LIN {X 0,Y 464.537,Z 936.315,A -85,B 0,C 180,E1 20832.687,E2 20832.687} C_VEL
LIN {X 0,Y 462.076,Z 957.618,A -85,B 0,C 180,E1 20831.71,E2 20831.71} C_VEL
LIN {X 0,Y 459.345,Z 978.775,A -85,B 0,C 180,E1 20830.531,E2 20830.531} C_VEL
LIN {X 0,Y 456.263,Z 999.373,A -85,B 0,C 180,E1 20829.127,E2 20829.127} C_VEL
LIN {X 0,Y 453.115,Z 1019.391,A -85,B 0,C 180,E1 20827.519,E2 20827.519} C_VEL
LIN {X 0,Y 449.993,Z 1037.958,A -85,B 0,C 180,E1 20825.758,E2 20825.758} C_VEL
LIN {X 0,Y 446.561,Z 1057.743,A -85,B 0,C 180,E1 20823.576,E2 20823.576} C_VEL
LIN {X 0,Y 443.731,Z 1074.21,A -85,B 0,C 180,E1 20821.464,E2 20821.464} C_VEL
LIN {X 0,Y 440.916,Z 1090.601,A -85,B 0,C 180,E1 20819.031,E2 20819.031} C_VEL
LIN {X 0,Y 438.586,Z 1105.226,A -85,B 0,C 180,E1 20816.54,E2 20816.54} C_VEL
LIN {X 0,Y 436.583,Z 1118.418,A -85,B 0,C 180,E1 20813.914,E2 20813.914} C_VEL
LIN {X 0,Y 434.957,Z 1130.257,A -85,B 0,C 180,E1 20811.156,E2 20811.156} C_VEL
LIN {X 0,Y 433.707,Z 1140.6,A -85,B 0,C 180,E1 20808.272,E2 20808.272} C_VEL
LIN {X 0,Y 432.808,Z 1149.992,A -85,B 0,C 180,E1 20805.132,E2 20805.132} C_VEL
LIN {X 0,Y 432.328,Z 1156.56,A -85,B 0,C 180,E1 20802.42,E2 20802.42} C_VEL
LIN {X 0,Y 432.052,Z 1162.429,A -85,B 0,C 180,E1 20799.322,E2 20799.322} C_VEL
LIN {X 0,Y 431.943,Z 1166.119,A -85,B 0,C 180,E1 20796.646,E2 20796.646} C_VEL
LIN {X 0,Y 431.895,Z 1168.848,A -85,B 0,C 180,E1 20793.583,E2 20793.583} C_VEL
LIN {X 0,Y 431.889,Z 1169.849,A -85,B 0,C 180,E1 20790.928,E2 20790.928} C_VEL
LIN {X 0,Y 431.905,Z 1169.689,A -85,B 0,C 180,E1 20788.142,E2 20788.142} C_VEL
LIN {X 0,Y 431.913,Z 1167.954,A -85,B 0,C 180,E1 20785.219,E2 20785.219} C_VEL
LIN {X 0,Y 431.957,Z 1165,A -85,B 0,C 180,E1 20782.418,E2 20782.418} C_VEL
LIN {X 0,Y 432.148,Z 1160.081,A -85,B 0,C 180,E1 20779.333,E2 20779.333} C_VEL
LIN {X 0,Y 432.493,Z 1154.133,A -85,B 0,C 180,E1 20776.497,E2 20776.497} C_VEL
LIN {X 0,Y 433.141,Z 1146.144,A -85,B 0,C 180,E1 20773.505,E2 20773.505} C_VEL
LIN {X 0,Y 434.129,Z 1136.928,A -85,B 0,C 180,E1 20770.631,E2 20770.631} C_VEL
LIN {X 0,Y 435.547,Z 1125.712,A -85,B 0,C 180,E1 20767.741,E2 20767.741} C_VEL
LIN {X 0,Y 437.273,Z 1113.83,A -85,B 0,C 180,E1 20765.119,E2 20765.119} C_VEL
LIN {X 0,Y 439.435,Z 1099.732,A -85,B 0,C 180,E1 20762.49,E2 20762.49} C_VEL
LIN {X 0,Y 442.212,Z 1082.982,A -85,B 0,C 180,E1 20759.795,E2 20759.795} C_VEL
LIN {X 0,Y 445.049,Z 1066.635,A -85,B 0,C 180,E1 20757.524,E2 20757.524} C_VEL
LIN {X 0,Y 448.073,Z 1049.082,A -85,B 0,C 180,E1 20755.427,E2 20755.427} C_VEL
LIN {X 0,Y 451.263,Z 1030.575,A -85,B 0,C 180,E1 20753.501,E2 20753.501} C_VEL
LIN {X 0,Y 454.405,Z 1011.335,A -85,B 0,C 180,E1 20751.807,E2 20751.807} C_VEL
LIN {X 0,Y 457.549,Z 991.207,A -85,B 0,C 180,E1 20750.282,E2 20750.282} C_VEL
LIN {X 0,Y 460.346,Z 970.958,A -85,B 0,C 180,E1 20749.009,E2 20749.009} C_VEL
LIN {X 0,Y 463.115,Z 948.971,A -85,B 0,C 180,E1 20747.862,E2 20747.862} C_VEL
LIN {X 0,Y 465.361,Z 927.596,A -85,B 0,C 180,E1 20746.986,E2 20746.986} C_VEL
LIN {X 0,Y 467.381,Z 903.992,A -85,B 0,C 180,E1 20746.249,E2 20746.249} C_VEL
LIN {X 0,Y 468.614,Z 882.183,A -85,B 0,C 180,E1 20745.765,E2 20745.765} C_VEL
LIN {X 0,Y 474.642,Z 683.276,A -85,B 0,C 180,E1 20742.249,E2 20742.249} C_VEL
LIN {X 0,Y 477.34,Z 594.822,A -85,B 0,C 180,E1 20740.649,E2 20740.649} C_VEL
LIN {X 0,Y 465.354,Z 575.94,A -85,B 0,C 180,E1 20738.463,E2 20738.463} C_VEL
LIN {X 0,Y 455.422,Z 561.586,A -85,B 0,C 180,E1 20736.51,E2 20736.51} C_VEL
LIN {X 0,Y 446.552,Z 549.244,A -85,B 0,C 180,E1 20734.622,E2 20734.622} C_VEL
LIN {X 0,Y 442.442,Z 543.776,A -85,B 0,C 180,E1 20733.696,E2 20733.696} C_VEL
LIN {X 0,Y 438.178,Z 538.303,A -85,B 0,C 180,E1 20732.699,E2 20732.699} C_VEL
LIN {X 0,Y 436.612,Z 536.106,A -85,B 0,C 180,E1 20732.247,E2 20732.247} C_VEL
LIN {X 0,Y 435.538,Z 533.777,A -85,B 0,C 180,E1 20731.716,E2 20731.716} C_VEL
LIN {X 0,Y 433.709,Z 530.877,A -85,B 0,C 180,E1 20730.937,E2 20730.937} C_VEL
LIN {X 0,Y 433.24,Z 529.049,A -85,B 0,C 180,E1 20730.552,E2 20730.552} C_VEL
LIN {X 0,Y 433.259,Z 529.072,A -85,B 0,C 180,E1 20726.892,E2 20726.892} C_VEL
LIN {X 0,Y 433.245,Z 529.031,A -85,B 0,C 180,E1 20723.099,E2 20723.099} C_VEL
LIN {X 0,Y 433.233,Z 529.057,A -85,B 0,C 180,E1 20719.41,E2 20719.41} C_VEL
LIN {X 0,Y 433.242,Z 529.06,A -85,B 0,C 180,E1 20715.528,E2 20715.528} C_VEL
LIN {X 0,Y 433.249,Z 529.036,A -85,B 0,C 180,E1 20711.852,E2 20711.852} C_VEL
LIN {X 0,Y 433.249,Z 529.074,A -85,B 0,C 180,E1 20708.083,E2 20708.083} C_VEL
LIN {X 0,Y 433.252,Z 529.078,A -85,B 0,C 180,E1 20704.235,E2 20704.235} C_VEL
LIN {X 0,Y 433.254,Z 529.079,A -85,B 0,C 180,E1 20700.396,E2 20700.396} C_VEL
LIN {X 0,Y 433.255,Z 529.08,A -85,B 0,C 180,E1 20696.56,E2 20696.56} C_VEL
LIN {X 0,Y 433.254,Z 529.079,A -85,B 0,C 180,E1 20692.708,E2 20692.708} C_VEL
LIN {X 0,Y 433.225,Z 529.03,A -85,B 0,C 180,E1 20688.956,E2 20688.956} C_VEL
LIN {X 0,Y 433.233,Z 529.076,A -85,B 0,C 180,E1 20685.156,E2 20685.156} C_VEL
LIN {X 0,Y 433.249,Z 529.036,A -85,B 0,C 180,E1 20681.429,E2 20681.429} C_VEL
LIN {X 0,Y 433.262,Z 529.045,A -85,B 0,C 180,E1 20677.618,E2 20677.618} C_VEL
LIN {X 0,Y 433.23,Z 529.076,A -85,B 0,C 180,E1 20673.844,E2 20673.844} C_VEL
LIN {X 0,Y 433.205,Z 529.041,A -85,B 0,C 180,E1 20670.096,E2 20670.096} C_VEL
LIN {X 0,Y 433.235,Z 529.287,A -85,B 0,C 180,E1 20668.028,E2 20668.028} C_VEL
LIN {X 0,Y 434.286,Z 532.203,A -85,B 0,C 180,E1 20667.715,E2 20667.715} C_VEL
LIN {X 0,Y 436.698,Z 534.701,A -85,B 0,C 180,E1 20667.137,E2 20667.137} C_VEL
LIN {X 0,Y 438.011,Z 535.73,A -85,B 0,C 180,E1 20666.838,E2 20666.838} C_VEL
LIN {X 0,Y 440.301,Z 539.399,A -85,B 0,C 180,E1 20666.274,E2 20666.274} C_VEL
LIN {X 0,Y 442.889,Z 541.924,A -85,B 0,C 180,E1 20665.698,E2 20665.698} C_VEL
LIN {X 0,Y 446.059,Z 546.162,A -85,B 0,C 180,E1 20664.982,E2 20664.982} C_VEL
LIN {X 0,Y 447.716,Z 548.187,A -85,B 0,C 180,E1 20664.622,E2 20664.622} C_VEL
LIN {X 0,Y 452.356,Z 554.185,A -85,B 0,C 180,E1 20663.635,E2 20663.635} C_VEL
LIN {X 0,Y 459.599,Z 563.567,A -85,B 0,C 180,E1 20662.177,E2 20662.177} C_VEL
LIN {X 0,Y 471.372,Z 579.87,A -85,B 0,C 180,E1 20659.97,E2 20659.97} C_VEL
LIN {X 0,Y 477.284,Z 588.789,A -85,B 0,C 180,E1 20658.922,E2 20658.922} C_VEL
LIN {X 0,Y 470.626,Z 800.468,A -85,B 0,C 180,E1 20655.158,E2 20655.158} C_VEL
LIN {X 0,Y 469.076,Z 852.641,A -85,B 0,C 180,E1 20654.242,E2 20654.242} C_VEL
LIN {X 0,Y 468.06,Z 860.337,A -85,B 0,C 180,E1 20654.186,E2 20654.186} C_VEL
LIN {X 0,Y 462.56,Z 879.729,A -85,B 0,C 180,E1 20654.257,E2 20654.257} C_VEL
LIN {X 0,Y 461.266,Z 887.24,A -85,B 0,C 180,E1 20654.119,E2 20654.119} C_VEL
LIN {X 0,Y 459.307,Z 908.693,A -85,B 0,C 180,E1 20653.361,E2 20653.361} C_VEL
LIN {X 0,Y 456.826,Z 930.04,A -85,B 0,C 180,E1 20652.387,E2 20652.387} C_VEL
LIN {X 0,Y 454.256,Z 949.055,A -85,B 0,C 180,E1 20651.325,E2 20651.325} C_VEL
LIN {X 0,Y 450.888,Z 970.761,A -85,B 0,C 180,E1 20649.857,E2 20649.857} C_VEL
LIN {X 0,Y 447.634,Z 990.006,A -85,B 0,C 180,E1 20648.305,E2 20648.305} C_VEL
LIN {X 0,Y 444.229,Z 1008.539,A -85,B 0,C 180,E1 20646.532,E2 20646.532} C_VEL
LIN {X 0,Y 440.839,Z 1026.51,A -85,B 0,C 180,E1 20644.543,E2 20644.543} C_VEL
LIN {X 0,Y 437.473,Z 1043.473,A -85,B 0,C 180,E1 20642.332,E2 20642.332} C_VEL
LIN {X 0,Y 434.444,Z 1059.247,A -85,B 0,C 180,E1 20639.962,E2 20639.962} C_VEL
LIN {X 0,Y 431.785,Z 1073.227,A -85,B 0,C 180,E1 20637.515,E2 20637.515} C_VEL
LIN {X 0,Y 429.287,Z 1087.359,A -85,B 0,C 180,E1 20634.64,E2 20634.64} C_VEL
LIN {X 0,Y 427.514,Z 1098.552,A -85,B 0,C 180,E1 20631.976,E2 20631.976} C_VEL
LIN {X 0,Y 425.953,Z 1109.995,A -85,B 0,C 180,E1 20628.759,E2 20628.759} C_VEL
LIN {X 0,Y 425.007,Z 1118.9,A -85,B 0,C 180,E1 20625.803,E2 20625.803} C_VEL
LIN {X 0,Y 424.409,Z 1125.853,A -85,B 0,C 180,E1 20622.933,E2 20622.933} C_VEL
LIN {X 0,Y 424.087,Z 1131.521,A -85,B 0,C 180,E1 20620.048,E2 20620.048} C_VEL
LIN {X 0,Y 423.938,Z 1135.585,A -85,B 0,C 180,E1 20617.181,E2 20617.181} C_VEL
LIN {X 0,Y 423.914,Z 1138.257,A -85,B 0,C 180,E1 20614.464,E2 20614.464} C_VEL
LIN {X 0,Y 423.907,Z 1139.772,A -85,B 0,C 180,E1 20611.352,E2 20611.352} C_VEL
LIN {X 0,Y 423.905,Z 1139.788,A -85,B 0,C 180,E1 20608.649,E2 20608.649} C_VEL
LIN {X 0,Y 423.911,Z 1138.333,A -85,B 0,C 180,E1 20605.536,E2 20605.536} C_VEL
LIN {X 0,Y 423.935,Z 1135.693,A -85,B 0,C 180,E1 20602.819,E2 20602.819} C_VEL
LIN {X 0,Y 424.081,Z 1131.671,A -85,B 0,C 180,E1 20599.952,E2 20599.952} C_VEL
LIN {X 0,Y 424.401,Z 1126.052,A -85,B 0,C 180,E1 20597.067,E2 20597.067} C_VEL
LIN {X 0,Y 425.034,Z 1118.689,A -85,B 0,C 180,E1 20594.024,E2 20594.024} C_VEL
LIN {X 0,Y 425.988,Z 1109.72,A -85,B 0,C 180,E1 20591.068,E2 20591.068} C_VEL
LIN {X 0,Y 427.62,Z 1097.777,A -85,B 0,C 180,E1 20587.742,E2 20587.742} C_VEL
LIN {X 0,Y 429.442,Z 1086.497,A -85,B 0,C 180,E1 20585.076,E2 20585.076} C_VEL
LIN {X 0,Y 431.907,Z 1072.551,A -85,B 0,C 180,E1 20582.27,E2 20582.27} C_VEL
LIN {X 0,Y 434.689,Z 1058.071,A -85,B 0,C 180,E1 20579.753,E2 20579.753} C_VEL
LIN {X 0,Y 437.749,Z 1042.06,A -85,B 0,C 180,E1 20577.381,E2 20577.381} C_VEL
LIN {X 0,Y 441.243,Z 1024.324,A -85,B 0,C 180,E1 20575.114,E2 20575.114} C_VEL
LIN {X 0,Y 444.47,Z 1007.272,A -85,B 0,C 180,E1 20573.246,E2 20573.246} C_VEL
LIN {X 0,Y 448.168,Z 986.861,A -85,B 0,C 180,E1 20571.338,E2 20571.338} C_VEL
LIN {X 0,Y 451.394,Z 967.84,A -85,B 0,C 180,E1 20569.835,E2 20569.835} C_VEL
LIN {X 0,Y 454.551,Z 946.907,A -85,B 0,C 180,E1 20568.456,E2 20568.456} C_VEL
LIN {X 0,Y 457.149,Z 927.589,A -85,B 0,C 180,E1 20567.396,E2 20567.396} C_VEL
LIN {X 0,Y 459.664,Z 904.799,A -85,B 0,C 180,E1 20566.396,E2 20566.396} C_VEL
LIN {X 0,Y 461.729,Z 881.961,A -85,B 0,C 180,E1 20565.628,E2 20565.628} C_VEL
LIN {X 0,Y 463.1,Z 859.095,A -85,B 0,C 180,E1 20565.097,E2 20565.097} C_VEL
LIN {X 0,Y 469.617,Z 660.74,A -85,B 0,C 180,E1 20561.547,E2 20561.547} C_VEL
LIN {X 0,Y 471.884,Z 592.324,A -85,B 0,C 180,E1 20560.3,E2 20560.3} C_VEL
LIN {X 0,Y 459.321,Z 574.267,A -85,B 0,C 180,E1 20557.949,E2 20557.949} C_VEL
LIN {X 0,Y 450.693,Z 562.894,A -85,B 0,C 180,E1 20556.205,E2 20556.205} C_VEL
LIN {X 0,Y 446.573,Z 557.588,A -85,B 0,C 180,E1 20555.325,E2 20555.325} C_VEL
LIN {X 0,Y 442.923,Z 552.874,A -85,B 0,C 180,E1 20554.514,E2 20554.514} C_VEL
LIN {X 0,Y 438.984,Z 547.828,A -85,B 0,C 180,E1 20553.606,E2 20553.606} C_VEL
LIN {X 0,Y 435.708,Z 543.956,A -85,B 0,C 180,E1 20552.83,E2 20552.83} C_VEL
LIN {X 0,Y 434.421,Z 542.142,A -85,B 0,C 180,E1 20552.508,E2 20552.508} C_VEL
LIN {X 0,Y 431.434,Z 539.099,A -85,B 0,C 180,E1 20551.78,E2 20551.78} C_VEL
LIN {X 0,Y 429.779,Z 536.292,A -85,B 0,C 180,E1 20551.33,E2 20551.33} C_VEL
LIN {X 0,Y 426.843,Z 533.857,A -85,B 0,C 180,E1 20550.591,E2 20550.591} C_VEL
LIN {X 0,Y 425.447,Z 530.984,A -85,B 0,C 180,E1 20550.173,E2 20550.173} C_VEL
LIN {X 0,Y 425.266,Z 530.032,A -85,B 0,C 180,E1 20550.092,E2 20550.092} C_VEL
LIN {X 0,Y 425.304,Z 530.071,A -85,B 0,C 180,E1 20546.38,E2 20546.38} C_VEL
LIN {X 0,Y 425.32,Z 530.023,A -85,B 0,C 180,E1 20542.5,E2 20542.5} C_VEL
LIN {X 0,Y 425.295,Z 530.039,A -85,B 0,C 180,E1 20538.789,E2 20538.789} C_VEL
LIN {X 0,Y 425.283,Z 530.05,A -85,B 0,C 180,E1 20534.988,E2 20534.988} C_VEL
LIN {X 0,Y 425.29,Z 530.064,A -85,B 0,C 180,E1 20531.115,E2 20531.115} C_VEL
LIN {X 0,Y 425.312,Z 530.065,A -85,B 0,C 180,E1 20527.294,E2 20527.294} C_VEL
LIN {X 0,Y 425.316,Z 530.066,A -85,B 0,C 180,E1 20523.505,E2 20523.505} C_VEL
LIN {X 0,Y 425.318,Z 530.068,A -85,B 0,C 180,E1 20519.596,E2 20519.596} C_VEL
LIN {X 0,Y 425.314,Z 530.071,A -85,B 0,C 180,E1 20515.686,E2 20515.686} C_VEL
LIN {X 0,Y 425.313,Z 530.068,A -85,B 0,C 180,E1 20511.778,E2 20511.778} C_VEL
LIN {X 0,Y 425.306,Z 530.02,A -85,B 0,C 180,E1 20507.923,E2 20507.923} C_VEL
LIN {X 0,Y 425.314,Z 530.047,A -85,B 0,C 180,E1 20504.175,E2 20504.175} C_VEL
LIN {X 0,Y 425.3,Z 530.048,A -85,B 0,C 180,E1 20500.356,E2 20500.356} C_VEL
LIN {X 0,Y 425.291,Z 530.026,A -85,B 0,C 180,E1 20496.475,E2 20496.475} C_VEL
LIN {X 0,Y 425.308,Z 530.055,A -85,B 0,C 180,E1 20492.703,E2 20492.703} C_VEL
LIN {X 0,Y 425.34,Z 530.158,A -85,B 0,C 180,E1 20491.037,E2 20491.037} C_VEL
LIN {X 0,Y 426.673,Z 533.637,A -85,B 0,C 180,E1 20490.212,E2 20490.212} C_VEL
LIN {X 0,Y 428.26,Z 535.701,A -85,B 0,C 180,E1 20489.561,E2 20489.561} C_VEL
LIN {X 0,Y 431.136,Z 539.923,A -85,B 0,C 180,E1 20488.742,E2 20488.742} C_VEL
LIN {X 0,Y 433.347,Z 542.697,A -85,B 0,C 180,E1 20488.183,E2 20488.183} C_VEL
LIN {X 0,Y 437.254,Z 547.799,A -85,B 0,C 180,E1 20487.224,E2 20487.224} C_VEL
LIN {X 0,Y 441.264,Z 553.084,A -85,B 0,C 180,E1 20486.28,E2 20486.28} C_VEL
LIN {X 0,Y 450.845,Z 566.205,A -85,B 0,C 180,E1 20484.163,E2 20484.163} C_VEL
LIN {X 0,Y 462.48,Z 583.389,A -85,B 0,C 180,E1 20481.807,E2 20481.807} C_VEL
LIN {X 0,Y 472.123,Z 598.819,A -85,B 0,C 180,E1 20479.998,E2 20479.998} C_VEL
LIN {X 0,Y 465.354,Z 804.742,A -85,B 0,C 180,E1 20476.303,E2 20476.303} C_VEL
LIN {X 0,Y 462.484,Z 890.625,A -85,B 0,C 180,E1 20474.758,E2 20474.758} C_VEL
LIN {X 0,Y 460.703,Z 913.95,A -85,B 0,C 180,E1 20474.154,E2 20474.154} C_VEL
LIN {X 0,Y 458.512,Z 936.783,A -85,B 0,C 180,E1 20473.343,E2 20473.343} C_VEL
LIN {X 0,Y 456,Z 957.431,A -85,B 0,C 180,E1 20472.387,E2 20472.387} C_VEL
LIN {X 0,Y 453.13,Z 978.557,A -85,B 0,C 180,E1 20471.199,E2 20471.199} C_VEL
LIN {X 0,Y 449.911,Z 998.994,A -85,B 0,C 180,E1 20469.794,E2 20469.794} C_VEL
LIN {X 0,Y 446.561,Z 1019.08,A -85,B 0,C 180,E1 20468.168,E2 20468.168} C_VEL
LIN {X 0,Y 443.253,Z 1037.646,A -85,B 0,C 180,E1 20466.388,E2 20466.388} C_VEL
LIN {X 0,Y 439.617,Z 1057.429,A -85,B 0,C 180,E1 20464.178,E2 20464.178} C_VEL
LIN {X 0,Y 436.566,Z 1074.041,A -85,B 0,C 180,E1 20462.019,E2 20462.019} C_VEL
LIN {X 0,Y 433.599,Z 1090.286,A -85,B 0,C 180,E1 20459.569,E2 20459.569} C_VEL
LIN {X 0,Y 431.097,Z 1104.912,A -85,B 0,C 180,E1 20457.038,E2 20457.038} C_VEL
LIN {X 0,Y 428.886,Z 1118.491,A -85,B 0,C 180,E1 20454.283,E2 20454.283} C_VEL
LIN {X 0,Y 427.144,Z 1130.699,A -85,B 0,C 180,E1 20451.418,E2 20451.418} C_VEL
LIN {X 0,Y 425.937,Z 1140.14,A -85,B 0,C 180,E1 20448.759,E2 20448.759} C_VEL
LIN {X 0,Y 424.967,Z 1149.285,A -85,B 0,C 180,E1 20445.698,E2 20445.698} C_VEL
LIN {X 0,Y 424.386,Z 1156.257,A -85,B 0,C 180,E1 20442.795,E2 20442.795} C_VEL
LIN {X 0,Y 424.062,Z 1162.223,A -85,B 0,C 180,E1 20439.637,E2 20439.637} C_VEL
LIN {X 0,Y 423.938,Z 1165.959,A -85,B 0,C 180,E1 20436.908,E2 20436.908} C_VEL
LIN {X 0,Y 423.909,Z 1168.732,A -85,B 0,C 180,E1 20433.883,E2 20433.883} C_VEL
LIN {X 0,Y 423.896,Z 1169.826,A -85,B 0,C 180,E1 20431.081,E2 20431.081} C_VEL
LIN {X 0,Y 423.905,Z 1169.735,A -85,B 0,C 180,E1 20428.378,E2 20428.378} C_VEL
LIN {X 0,Y 423.912,Z 1168.067,A -85,B 0,C 180,E1 20425.264,E2 20425.264} C_VEL
LIN {X 0,Y 423.95,Z 1165.319,A -85,B 0,C 180,E1 20422.547,E2 20422.547} C_VEL
LIN {X 0,Y 424.145,Z 1160.589,A -85,B 0,C 180,E1 20419.404,E2 20419.404} C_VEL
LIN {X 0,Y 424.487,Z 1154.934,A -85,B 0,C 180,E1 20416.604,E2 20416.604} C_VEL
LIN {X 0,Y 425.182,Z 1146.952,A -85,B 0,C 180,E1 20413.468,E2 20413.468} C_VEL
LIN {X 0,Y 426.155,Z 1138.306,A -85,B 0,C 180,E1 20410.681,E2 20410.681} C_VEL
LIN {X 0,Y 427.604,Z 1127.286,A -85,B 0,C 180,E1 20407.74,E2 20407.74} C_VEL
LIN {X 0,Y 429.363,Z 1115.512,A -85,B 0,C 180,E1 20405.07,E2 20405.07} C_VEL
LIN {X 0,Y 431.603,Z 1101.771,A -85,B 0,C 180,E1 20402.398,E2 20402.398} C_VEL
LIN {X 0,Y 434.258,Z 1086.845,A -85,B 0,C 180,E1 20399.871,E2 20399.871} C_VEL
LIN {X 0,Y 437.209,Z 1070.436,A -85,B 0,C 180,E1 20397.491,E2 20397.491} C_VEL
LIN {X 0,Y 440.547,Z 1052.605,A -85,B 0,C 180,E1 20395.243,E2 20395.243} C_VEL
LIN {X 0,Y 443.726,Z 1034.931,A -85,B 0,C 180,E1 20393.335,E2 20393.335} C_VEL
LIN {X 0,Y 447.379,Z 1014.302,A -85,B 0,C 180,E1 20391.424,E2 20391.424} C_VEL
LIN {X 0,Y 450.413,Z 995.966,A -85,B 0,C 180,E1 20389.982,E2 20389.982} C_VEL
LIN {X 0,Y 453.761,Z 973.851,A -85,B 0,C 180,E1 20388.519,E2 20388.519} C_VEL
LIN {X 0,Y 456.604,Z 952.693,A -85,B 0,C 180,E1 20387.371,E2 20387.371} C_VEL
LIN {X 0,Y 459.196,Z 929.901,A -85,B 0,C 180,E1 20386.393,E2 20386.393} C_VEL
LIN {X 0,Y 461.34,Z 907.273,A -85,B 0,C 180,E1 20385.648,E2 20385.648} C_VEL
LIN {X 0,Y 462.784,Z 883.982,A -85,B 0,C 180,E1 20385.112,E2 20385.112} C_VEL
LIN {X 0,Y 469.117,Z 687.272,A -85,B 0,C 180,E1 20381.598,E2 20381.598} C_VEL
LIN {X 0,Y 472.018,Z 598.678,A -85,B 0,C 180,E1 20379.988,E2 20379.988} C_VEL
LIN {X 0,Y 460.697,Z 580.715,A -85,B 0,C 180,E1 20377.854,E2 20377.854} C_VEL
LIN {X 0,Y 449.263,Z 564.004,A -85,B 0,C 180,E1 20375.511,E2 20375.511} C_VEL
LIN {X 0,Y 439.388,Z 550.524,A -85,B 0,C 180,E1 20373.297,E2 20373.297} C_VEL
LIN {X 0,Y 431.55,Z 540.339,A -85,B 0,C 180,E1 20371.38,E2 20371.38} C_VEL
LIN {X 0,Y 428.411,Z 536.179,A -85,B 0,C 180,E1 20370.56,E2 20370.56} C_VEL
LIN {X 0,Y 427.612,Z 534.749,A -85,B 0,C 180,E1 20370.18,E2 20370.18} C_VEL
LIN {X 0,Y 425.837,Z 532.067,A -85,B 0,C 180,E1 20369.388,E2 20369.388} C_VEL
LIN {X 0,Y 425.321,Z 530.02,A -85,B 0,C 180,E1 20368.913,E2 20368.913} C_VEL
LIN {X 0,Y 425.306,Z 530.033,A -85,B 0,C 180,E1 20365.161,E2 20365.161} C_VEL
LIN {X 0,Y 425.296,Z 530.06,A -85,B 0,C 180,E1 20361.37,E2 20361.37} C_VEL
LIN {X 0,Y 425.293,Z 530.015,A -85,B 0,C 180,E1 20357.513,E2 20357.513} C_VEL
LIN {X 0,Y 425.32,Z 530.067,A -85,B 0,C 180,E1 20353.735,E2 20353.735} C_VEL
LIN {X 0,Y 425.307,Z 530.02,A -85,B 0,C 180,E1 20349.881,E2 20349.881} C_VEL
LIN {X 0,Y 425.312,Z 530.057,A -85,B 0,C 180,E1 20346.047,E2 20346.047} C_VEL
LIN {X 0,Y 425.313,Z 530.057,A -85,B 0,C 180,E1 20342.155,E2 20342.155} C_VEL
LIN {X 0,Y 425.314,Z 530.056,A -85,B 0,C 180,E1 20338.383,E2 20338.383} C_VEL
LIN {X 0,Y 425.315,Z 530.055,A -85,B 0,C 180,E1 20334.469,E2 20334.469} C_VEL
LIN {X 0,Y 425.297,Z 530.03,A -85,B 0,C 180,E1 20330.801,E2 20330.801} C_VEL
LIN {X 0,Y 425.29,Z 530.057,A -85,B 0,C 180,E1 20326.956,E2 20326.956} C_VEL
LIN {X 0,Y 425.293,Z 530.018,A -85,B 0,C 180,E1 20323.191,E2 20323.191} C_VEL
LIN {X 0,Y 425.318,Z 530.071,A -85,B 0,C 180,E1 20319.333,E2 20319.333} C_VEL
LIN {X 0,Y 425.314,Z 530.02,A -85,B 0,C 180,E1 20315.477,E2 20315.477} C_VEL
LIN {X 0,Y 425.283,Z 530.041,A -85,B 0,C 180,E1 20311.799,E2 20311.799} C_VEL
LIN {X 0,Y 425.288,Z 530.141,A -85,B 0,C 180,E1 20309.779,E2 20309.779} C_VEL
LIN {X 0,Y 426.312,Z 533.057,A -85,B 0,C 180,E1 20309.445,E2 20309.445} C_VEL
LIN {X 0,Y 428.949,Z 535.811,A -85,B 0,C 180,E1 20308.759,E2 20308.759} C_VEL
LIN {X 0,Y 430.205,Z 536.766,A -85,B 0,C 180,E1 20308.451,E2 20308.451} C_VEL
LIN {X 0,Y 432.502,Z 540.463,A -85,B 0,C 180,E1 20307.839,E2 20307.839} C_VEL
LIN {X 0,Y 435.168,Z 543.011,A -85,B 0,C 180,E1 20307.203,E2 20307.203} C_VEL
LIN {X 0,Y 438.268,Z 547.184,A -85,B 0,C 180,E1 20306.45,E2 20306.45} C_VEL
LIN {X 0,Y 440.006,Z 549.062,A -85,B 0,C 180,E1 20306.052,E2 20306.052} C_VEL
LIN {X 0,Y 443.612,Z 553.549,A -85,B 0,C 180,E1 20305.233,E2 20305.233} C_VEL
LIN {X 0,Y 455.899,Z 569.668,A -85,B 0,C 180,E1 20302.63,E2 20302.63} C_VEL
LIN {X 0,Y 468.601,Z 587.464,A -85,B 0,C 180,E1 20300.2,E2 20300.2} C_VEL
LIN {X 0,Y 471.942,Z 592.711,A -85,B 0,C 180,E1 20299.589,E2 20299.589} C_VEL
LIN {X 0,Y 464.942,Z 803.271,A -85,B 0,C 180,E1 20295.813,E2 20295.813} C_VEL
LIN {X 0,Y 462.728,Z 867.077,A -85,B 0,C 180,E1 20294.654,E2 20294.654} C_VEL
LIN {X 0,Y 461.266,Z 887.24,A -85,B 0,C 180,E1 20294.119,E2 20294.119} C_VEL
LIN {X 0,Y 460.093,Z 893.703,A -85,B 0,C 180,E1 20293.996,E2 20293.996} C_VEL
LIN {X 0,Y 453.602,Z 914.002,A -85,B 0,C 180,E1 20293.769,E2 20293.769} C_VEL
LIN {X 0,Y 452.057,Z 921.17,A -85,B 0,C 180,E1 20293.529,E2 20293.529} C_VEL
LIN {X 0,Y 448.947,Z 944.218,A -85,B 0,C 180,E1 20292.319,E2 20292.319} C_VEL
LIN {X 0,Y 445.944,Z 963.696,A -85,B 0,C 180,E1 20291.068,E2 20291.068} C_VEL
LIN {X 0,Y 442.428,Z 983.9,A -85,B 0,C 180,E1 20289.508,E2 20289.508} C_VEL
LIN {X 0,Y 439.028,Z 1002.059,A -85,B 0,C 180,E1 20287.863,E2 20287.863} C_VEL
LIN {X 0,Y 435.258,Z 1020.828,A -85,B 0,C 180,E1 20285.859,E2 20285.859} C_VEL
LIN {X 0,Y 431.719,Z 1038.298,A -85,B 0,C 180,E1 20283.689,E2 20283.689} C_VEL
LIN {X 0,Y 428.36,Z 1054.211,A -85,B 0,C 180,E1 20281.368,E2 20281.368} C_VEL
LIN {X 0,Y 425.182,Z 1069.982,A -85,B 0,C 180,E1 20278.7,E2 20278.7} C_VEL
LIN {X 0,Y 422.625,Z 1083.118,A -85,B 0,C 180,E1 20276.107,E2 20276.107} C_VEL
LIN {X 0,Y 420.301,Z 1096.061,A -85,B 0,C 180,E1 20273.112,E2 20273.112} C_VEL
LIN {X 0,Y 418.633,Z 1106.867,A -85,B 0,C 180,E1 20270.176,E2 20270.176} C_VEL
LIN {X 0,Y 417.399,Z 1116.077,A -85,B 0,C 180,E1 20267.136,E2 20267.136} C_VEL
LIN {X 0,Y 416.568,Z 1124.643,A -85,B 0,C 180,E1 20263.747,E2 20263.747} C_VEL
LIN {X 0,Y 416.197,Z 1130.253,A -85,B 0,C 180,E1 20260.941,E2 20260.941} C_VEL
LIN {X 0,Y 415.977,Z 1135.107,A -85,B 0,C 180,E1 20257.736,E2 20257.736} C_VEL
LIN {X 0,Y 415.918,Z 1137.916,A -85,B 0,C 180,E1 20254.965,E2 20254.965} C_VEL
LIN {X 0,Y 415.905,Z 1139.682,A -85,B 0,C 180,E1 20251.929,E2 20251.929} C_VEL
LIN {X 0,Y 415.888,Z 1139.856,A -85,B 0,C 180,E1 20249.036,E2 20249.036} C_VEL
LIN {X 0,Y 415.9,Z 1138.87,A -85,B 0,C 180,E1 20246.279,E2 20246.279} C_VEL
LIN {X 0,Y 415.937,Z 1136.171,A -85,B 0,C 180,E1 20243.097,E2 20243.097} C_VEL
LIN {X 0,Y 416.063,Z 1132.703,A -85,B 0,C 180,E1 20240.456,E2 20240.456} C_VEL
LIN {X 0,Y 416.39,Z 1126.959,A -85,B 0,C 180,E1 20237.237,E2 20237.237} C_VEL
LIN {X 0,Y 416.946,Z 1120.455,A -85,B 0,C 180,E1 20234.42,E2 20234.42} C_VEL
LIN {X 0,Y 418.067,Z 1110.927,A -85,B 0,C 180,E1 20231.019,E2 20231.019} C_VEL
LIN {X 0,Y 419.56,Z 1100.834,A -85,B 0,C 180,E1 20228.028,E2 20228.028} C_VEL
LIN {X 0,Y 421.487,Z 1089.292,A -85,B 0,C 180,E1 20225.173,E2 20225.173} C_VEL
LIN {X 0,Y 423.891,Z 1076.638,A -85,B 0,C 180,E1 20222.463,E2 20222.463} C_VEL
LIN {X 0,Y 426.738,Z 1062.154,A -85,B 0,C 180,E1 20219.835,E2 20219.835} C_VEL
LIN {X 0,Y 430.204,Z 1045.359,A -85,B 0,C 180,E1 20217.212,E2 20217.212} C_VEL
LIN {X 0,Y 433.591,Z 1029.105,A -85,B 0,C 180,E1 20215.038,E2 20215.038} C_VEL
LIN {X 0,Y 437.304,Z 1010.733,A -85,B 0,C 180,E1 20212.936,E2 20212.936} C_VEL
LIN {X 0,Y 440.968,Z 991.968,A -85,B 0,C 180,E1 20211.092,E2 20211.092} C_VEL
LIN {X 0,Y 444.514,Z 972.038,A -85,B 0,C 180,E1 20209.454,E2 20209.454} C_VEL
LIN {X 0,Y 447.962,Z 951.174,A -85,B 0,C 180,E1 20208.01,E2 20208.01} C_VEL
LIN {X 0,Y 450.726,Z 931.709,A -85,B 0,C 180,E1 20206.902,E2 20206.902} C_VEL
LIN {X 0,Y 453.396,Z 910.155,A -85,B 0,C 180,E1 20205.896,E2 20205.896} C_VEL
LIN {X 0,Y 455.502,Z 888.157,A -85,B 0,C 180,E1 20205.107,E2 20205.107} C_VEL
LIN {X 0,Y 457.232,Z 864.174,A -85,B 0,C 180,E1 20204.485,E2 20204.485} C_VEL
LIN {X 0,Y 463.582,Z 682.197,A -85,B 0,C 180,E1 20201.19,E2 20201.19} C_VEL
LIN {X 0,Y 466.625,Z 596.426,A -85,B 0,C 180,E1 20199.623,E2 20199.623} C_VEL
LIN {X 0,Y 455.536,Z 580.349,A -85,B 0,C 180,E1 20197.484,E2 20197.484} C_VEL
LIN {X 0,Y 447.152,Z 569.143,A -85,B 0,C 180,E1 20195.745,E2 20195.745} C_VEL
LIN {X 0,Y 439.732,Z 559.486,A -85,B 0,C 180,E1 20194.09,E2 20194.09} C_VEL
LIN {X 0,Y 435.837,Z 554.527,A -85,B 0,C 180,E1 20193.172,E2 20193.172} C_VEL
LIN {X 0,Y 432.279,Z 549.967,A -85,B 0,C 180,E1 20192.297,E2 20192.297} C_VEL
LIN {X 0,Y 428.198,Z 545.337,A -85,B 0,C 180,E1 20191.267,E2 20191.267} C_VEL
LIN {X 0,Y 426.976,Z 543.425,A -85,B 0,C 180,E1 20190.931,E2 20190.931} C_VEL
LIN {X 0,Y 423.78,Z 540.286,A -85,B 0,C 180,E1 20190.091,E2 20190.091} C_VEL
LIN {X 0,Y 422.113,Z 537.382,A -85,B 0,C 180,E1 20189.596,E2 20189.596} C_VEL
LIN {X 0,Y 419.203,Z 535.18,A -85,B 0,C 180,E1 20188.803,E2 20188.803} C_VEL
LIN {X 0,Y 417.615,Z 532.313,A -85,B 0,C 180,E1 20188.298,E2 20188.298} C_VEL
LIN {X 0,Y 417.336,Z 531.023,A -85,B 0,C 180,E1 20188.157,E2 20188.157} C_VEL
LIN {X 0,Y 417.371,Z 531.011,A -85,B 0,C 180,E1 20184.449,E2 20184.449} C_VEL
LIN {X 0,Y 417.376,Z 531.057,A -85,B 0,C 180,E1 20180.619,E2 20180.619} C_VEL
LIN {X 0,Y 417.347,Z 531.003,A -85,B 0,C 180,E1 20176.851,E2 20176.851} C_VEL
LIN {X 0,Y 417.348,Z 531.058,A -85,B 0,C 180,E1 20173.015,E2 20173.015} C_VEL
LIN {X 0,Y 417.356,Z 531.052,A -85,B 0,C 180,E1 20169.098,E2 20169.098} C_VEL
LIN {X 0,Y 417.376,Z 531.046,A -85,B 0,C 180,E1 20165.361,E2 20165.361} C_VEL
LIN {X 0,Y 417.376,Z 531.044,A -85,B 0,C 180,E1 20161.51,E2 20161.51} C_VEL
LIN {X 0,Y 417.375,Z 531.044,A -85,B 0,C 180,E1 20157.666,E2 20157.666} C_VEL
LIN {X 0,Y 417.372,Z 531.044,A -85,B 0,C 180,E1 20153.812,E2 20153.812} C_VEL
LIN {X 0,Y 417.366,Z 531.012,A -85,B 0,C 180,E1 20149.929,E2 20149.929} C_VEL
LIN {X 0,Y 417.378,Z 531.055,A -85,B 0,C 180,E1 20145.979,E2 20145.979} C_VEL
LIN {X 0,Y 417.366,Z 531.006,A -85,B 0,C 180,E1 20142.143,E2 20142.143} C_VEL
LIN {X 0,Y 417.357,Z 531.047,A -85,B 0,C 180,E1 20138.35,E2 20138.35} C_VEL
LIN {X 0,Y 417.356,Z 531.037,A -85,B 0,C 180,E1 20134.455,E2 20134.455} C_VEL
LIN {X 0,Y 417.38,Z 531.084,A -85,B 0,C 180,E1 20132.824,E2 20132.824} C_VEL
LIN {X 0,Y 418.414,Z 534.136,A -85,B 0,C 180,E1 20132.072,E2 20132.072} C_VEL
LIN {X 0,Y 420.655,Z 536.651,A -85,B 0,C 180,E1 20131.267,E2 20131.267} C_VEL
LIN {X 0,Y 423.521,Z 540.811,A -85,B 0,C 180,E1 20130.435,E2 20130.435} C_VEL
LIN {X 0,Y 425.545,Z 542.984,A -85,B 0,C 180,E1 20129.892,E2 20129.892} C_VEL
LIN {X 0,Y 429.034,Z 547.532,A -85,B 0,C 180,E1 20128.962,E2 20128.962} C_VEL
LIN {X 0,Y 438.092,Z 559.651,A -85,B 0,C 180,E1 20126.709,E2 20126.709} C_VEL
LIN {X 0,Y 447.799,Z 573.224,A -85,B 0,C 180,E1 20124.512,E2 20124.512} C_VEL
LIN {X 0,Y 458.587,Z 589.268,A -85,B 0,C 180,E1 20122.277,E2 20122.277} C_VEL
LIN {X 0,Y 466.837,Z 602.668,A -85,B 0,C 180,E1 20120.68,E2 20120.68} C_VEL
LIN {X 0,Y 459.498,Z 814.285,A -85,B 0,C 180,E1 20116.853,E2 20116.853} C_VEL
LIN {X 0,Y 456.79,Z 890.66,A -85,B 0,C 180,E1 20115.462,E2 20115.462} C_VEL
LIN {X 0,Y 454.91,Z 914.036,A -85,B 0,C 180,E1 20114.85,E2 20114.85} C_VEL
LIN {X 0,Y 452.638,Z 936.485,A -85,B 0,C 180,E1 20114.049,E2 20114.049} C_VEL
LIN {X 0,Y 450.022,Z 957,A -85,B 0,C 180,E1 20113.094,E2 20113.094} C_VEL
LIN {X 0,Y 446.989,Z 978.269,A -85,B 0,C 180,E1 20111.89,E2 20111.89} C_VEL
LIN {X 0,Y 443.613,Z 998.688,A -85,B 0,C 180,E1 20110.475,E2 20110.475} C_VEL
LIN {X 0,Y 440.075,Z 1018.77,A -85,B 0,C 180,E1 20108.835,E2 20108.835} C_VEL
LIN {X 0,Y 436.565,Z 1037.333,A -85,B 0,C 180,E1 20107.038,E2 20107.038} C_VEL
LIN {X 0,Y 432.73,Z 1057.116,A -85,B 0,C 180,E1 20104.8,E2 20104.8} C_VEL
LIN {X 0,Y 429.462,Z 1073.777,A -85,B 0,C 180,E1 20102.605,E2 20102.605} C_VEL
LIN {X 0,Y 426.326,Z 1089.972,A -85,B 0,C 180,E1 20100.125,E2 20100.125} C_VEL
LIN {X 0,Y 423.641,Z 1104.597,A -85,B 0,C 180,E1 20097.554,E2 20097.554} C_VEL
LIN {X 0,Y 421.334,Z 1117.79,A -85,B 0,C 180,E1 20094.837,E2 20094.837} C_VEL
LIN {X 0,Y 419.485,Z 1129.86,A -85,B 0,C 180,E1 20091.976,E2 20091.976} C_VEL
LIN {X 0,Y 418.051,Z 1140.438,A -85,B 0,C 180,E1 20088.982,E2 20088.982} C_VEL
LIN {X 0,Y 417.066,Z 1149.329,A -85,B 0,C 180,E1 20085.985,E2 20085.985} C_VEL
LIN {X 0,Y 416.437,Z 1156.257,A -85,B 0,C 180,E1 20083.043,E2 20083.043} C_VEL
LIN {X 0,Y 416.074,Z 1162.223,A -85,B 0,C 180,E1 20079.824,E2 20079.824} C_VEL
LIN {X 0,Y 415.937,Z 1165.959,A -85,B 0,C 180,E1 20077.042,E2 20077.042} C_VEL
LIN {X 0,Y 415.912,Z 1168.712,A -85,B 0,C 180,E1 20073.997,E2 20073.997} C_VEL
LIN {X 0,Y 415.897,Z 1169.825,A -85,B 0,C 180,E1 20071.102,E2 20071.102} C_VEL
LIN {X 0,Y 415.905,Z 1169.734,A -85,B 0,C 180,E1 20068.347,E2 20068.347} C_VEL
LIN {X 0,Y 415.914,Z 1168.067,A -85,B 0,C 180,E1 20065.173,E2 20065.173} C_VEL
LIN {X 0,Y 415.96,Z 1165.319,A -85,B 0,C 180,E1 20062.403,E2 20062.403} C_VEL
LIN {X 0,Y 416.176,Z 1160.589,A -85,B 0,C 180,E1 20059.199,E2 20059.199} C_VEL
LIN {X 0,Y 416.536,Z 1155.042,A -85,B 0,C 180,E1 20056.394,E2 20056.394} C_VEL
LIN {X 0,Y 417.297,Z 1146.943,A -85,B 0,C 180,E1 20053.146,E2 20053.146} C_VEL
LIN {X 0,Y 418.313,Z 1138.224,A -85,B 0,C 180,E1 20050.345,E2 20050.345} C_VEL
LIN {X 0,Y 419.883,Z 1126.973,A -85,B 0,C 180,E1 20047.308,E2 20047.308} C_VEL
LIN {X 0,Y 421.791,Z 1115.131,A -85,B 0,C 180,E1 20044.576,E2 20044.576} C_VEL
LIN {X 0,Y 424.239,Z 1101.153,A -85,B 0,C 180,E1 20041.817,E2 20041.817} C_VEL
LIN {X 0,Y 427.181,Z 1085.644,A -85,B 0,C 180,E1 20039.163,E2 20039.163} C_VEL
LIN {X 0,Y 430.374,Z 1069.093,A -85,B 0,C 180,E1 20036.75,E2 20036.75} C_VEL
LIN {X 0,Y 434.02,Z 1050.515,A -85,B 0,C 180,E1 20034.41,E2 20034.41} C_VEL
LIN {X 0,Y 437.485,Z 1032.549,A -85,B 0,C 180,E1 20032.471,E2 20032.471} C_VEL
LIN {X 0,Y 441.278,Z 1012.057,A -85,B 0,C 180,E1 20030.591,E2 20030.591} C_VEL
LIN {X 0,Y 444.669,Z 992.571,A -85,B 0,C 180,E1 20029.069,E2 20029.069} C_VEL
LIN {X 0,Y 447.944,Z 971.476,A -85,B 0,C 180,E1 20027.702,E2 20027.702} C_VEL
LIN {X 0,Y 451.013,Z 949.828,A -85,B 0,C 180,E1 20026.543,E2 20026.543} C_VEL
LIN {X 0,Y 453.54,Z 928.064,A -85,B 0,C 180,E1 20025.631,E2 20025.631} C_VEL
LIN {X 0,Y 455.723,Z 905.485,A -85,B 0,C 180,E1 20024.901,E2 20024.901} C_VEL
LIN {X 0,Y 457.162,Z 882.708,A -85,B 0,C 180,E1 20024.381,E2 20024.381} C_VEL
LIN {X 0,Y 463.878,Z 684.959,A -85,B 0,C 180,E1 20020.818,E2 20020.818} C_VEL
LIN {X 0,Y 466.701,Z 602.401,A -85,B 0,C 180,E1 20019.299,E2 20019.299} C_VEL
LIN {X 0,Y 455.825,Z 585.122,A -85,B 0,C 180,E1 20017.179,E2 20017.179} C_VEL
LIN {X 0,Y 444.476,Z 568.386,A -85,B 0,C 180,E1 20014.767,E2 20014.767} C_VEL
LIN {X 0,Y 435.869,Z 556.703,A -85,B 0,C 180,E1 20012.777,E2 20012.777} C_VEL
LIN {X 0,Y 428.737,Z 547.24,A -85,B 0,C 180,E1 20010.984,E2 20010.984} C_VEL
LIN {X 0,Y 425.376,Z 542.692,A -85,B 0,C 180,E1 20010.082,E2 20010.082} C_VEL
LIN {X 0,Y 421.502,Z 538.211,A -85,B 0,C 180,E1 20009.019,E2 20009.019} C_VEL
LIN {X 0,Y 420.257,Z 536.218,A -85,B 0,C 180,E1 20008.646,E2 20008.646} C_VEL
LIN {X 0,Y 418.049,Z 533.449,A -85,B 0,C 180,E1 20007.755,E2 20007.755} C_VEL
LIN {X 0,Y 417.373,Z 531.039,A -85,B 0,C 180,E1 20007.175,E2 20007.175} C_VEL
LIN {X 0,Y 417.358,Z 531.004,A -85,B 0,C 180,E1 20003.283,E2 20003.283} C_VEL
LIN {X 0,Y 417.356,Z 531.03,A -85,B 0,C 180,E1 19999.451,E2 19999.451} C_VEL
LIN {X 0,Y 417.364,Z 531.031,A -85,B 0,C 180,E1 19995.563,E2 19995.563} C_VEL
LIN {X 0,Y 417.371,Z 531.007,A -85,B 0,C 180,E1 19991.749,E2 19991.749} C_VEL
LIN {X 0,Y 417.372,Z 531.055,A -85,B 0,C 180,E1 19987.848,E2 19987.848} C_VEL
LIN {X 0,Y 417.371,Z 531.06,A -85,B 0,C 180,E1 19983.983,E2 19983.983} C_VEL
LIN {X 0,Y 417.387,Z 531.059,A -85,B 0,C 180,E1 19980.137,E2 19980.137} C_VEL
LIN {X 0,Y 417.376,Z 531.057,A -85,B 0,C 180,E1 19976.154,E2 19976.154} C_VEL
LIN {X 0,Y 417.38,Z 531.052,A -85,B 0,C 180,E1 19972.29,E2 19972.29} C_VEL
LIN {X 0,Y 417.367,Z 531.006,A -85,B 0,C 180,E1 19968.391,E2 19968.391} C_VEL
LIN {X 0,Y 417.349,Z 531.04,A -85,B 0,C 180,E1 19964.72,E2 19964.72} C_VEL
LIN {X 0,Y 417.345,Z 531.025,A -85,B 0,C 180,E1 19960.839,E2 19960.839} C_VEL
LIN {X 0,Y 417.368,Z 531.012,A -85,B 0,C 180,E1 19957.164,E2 19957.164} C_VEL
LIN {X 0,Y 417.383,Z 531.059,A -85,B 0,C 180,E1 19953.233,E2 19953.233} C_VEL
LIN {X 0,Y 417.376,Z 531.216,A -85,B 0,C 180,E1 19951.684,E2 19951.684} C_VEL
LIN {X 0,Y 418.476,Z 534.17,A -85,B 0,C 180,E1 19951.298,E2 19951.298} C_VEL
LIN {X 0,Y 421.078,Z 536.837,A -85,B 0,C 180,E1 19950.559,E2 19950.559} C_VEL
LIN {X 0,Y 422.446,Z 537.789,A -85,B 0,C 180,E1 19950.196,E2 19950.196} C_VEL
LIN {X 0,Y 424.674,Z 541.411,A -85,B 0,C 180,E1 19949.55,E2 19949.55} C_VEL
LIN {X 0,Y 427.5,Z 544.113,A -85,B 0,C 180,E1 19948.817,E2 19948.817} C_VEL
LIN {X 0,Y 430.392,Z 548.099,A -85,B 0,C 180,E1 19948.055,E2 19948.055} C_VEL
LIN {X 0,Y 432.418,Z 550.215,A -85,B 0,C 180,E1 19947.558,E2 19947.558} C_VEL
LIN {X 0,Y 435.997,Z 554.676,A -85,B 0,C 180,E1 19946.685,E2 19946.685} C_VEL
LIN {X 0,Y 442.381,Z 562.951,A -85,B 0,C 180,E1 19945.201,E2 19945.201} C_VEL
LIN {X 0,Y 450.322,Z 573.28,A -85,B 0,C 180,E1 19943.484,E2 19943.484} C_VEL
LIN {X 0,Y 460.037,Z 586.826,A -85,B 0,C 180,E1 19941.527,E2 19941.527} C_VEL
LIN {X 0,Y 466.664,Z 596.689,A -85,B 0,C 180,E1 19940.269,E2 19940.269} C_VEL
LIN {X 0,Y 459.319,Z 806.086,A -85,B 0,C 180,E1 19936.484,E2 19936.484} C_VEL
LIN {X 0,Y 457.064,Z 867.537,A -85,B 0,C 180,E1 19935.356,E2 19935.356} C_VEL
LIN {X 0,Y 455.351,Z 889.873,A -85,B 0,C 180,E1 19934.746,E2 19934.746} C_VEL
LIN {X 0,Y 453.197,Z 911.996,A -85,B 0,C 180,E1 19933.937,E2 19933.937} C_VEL
LIN {X 0,Y 452.057,Z 921.17,A -85,B 0,C 180,E1 19933.529,E2 19933.529} C_VEL
LIN {X 0,Y 450.438,Z 928.516,A -85,B 0,C 180,E1 19933.271,E2 19933.271} C_VEL
LIN {X 0,Y 443.471,Z 946.981,A -85,B 0,C 180,E1 19932.795,E2 19932.795} C_VEL
LIN {X 0,Y 441.573,Z 953.973,A -85,B 0,C 180,E1 19932.443,E2 19932.443} C_VEL
LIN {X 0,Y 438.052,Z 974.061,A -85,B 0,C 180,E1 19931.013,E2 19931.013} C_VEL
LIN {X 0,Y 434.19,Z 994.384,A -85,B 0,C 180,E1 19929.293,E2 19929.293} C_VEL
LIN {X 0,Y 430.631,Z 1011.765,A -85,B 0,C 180,E1 19927.553,E2 19927.553} C_VEL
LIN {X 0,Y 426.591,Z 1030.63,A -85,B 0,C 180,E1 19925.348,E2 19925.348} C_VEL
LIN {X 0,Y 423.087,Z 1046.6,A -85,B 0,C 180,E1 19923.168,E2 19923.168} C_VEL
LIN {X 0,Y 419.633,Z 1062.37,A -85,B 0,C 180,E1 19920.658,E2 19920.658} C_VEL
LIN {X 0,Y 416.648,Z 1076.504,A -85,B 0,C 180,E1 19918.058,E2 19918.058} C_VEL
LIN {X 0,Y 414.06,Z 1089.232,A -85,B 0,C 180,E1 19915.304,E2 19915.304} C_VEL
LIN {X 0,Y 411.958,Z 1100.93,A -85,B 0,C 180,E1 19912.373,E2 19912.373} C_VEL
LIN {X 0,Y 410.334,Z 1110.961,A -85,B 0,C 180,E1 19909.354,E2 19909.354} C_VEL
LIN {X 0,Y 409.177,Z 1119.808,A -85,B 0,C 180,E1 19906.175,E2 19906.175} C_VEL
LIN {X 0,Y 408.478,Z 1126.566,A -85,B 0,C 180,E1 19903.159,E2 19903.159} C_VEL
LIN {X 0,Y 408.075,Z 1132.57,A -85,B 0,C 180,E1 19899.734,E2 19899.734} C_VEL
LIN {X 0,Y 407.937,Z 1136.066,A -85,B 0,C 180,E1 19897.04,E2 19897.04} C_VEL
LIN {X 0,Y 407.912,Z 1138.757,A -85,B 0,C 180,E1 19893.936,E2 19893.936} C_VEL
LIN {X 0,Y 407.901,Z 1139.818,A -85,B 0,C 180,E1 19891.124,E2 19891.124} C_VEL
LIN {X 0,Y 407.905,Z 1139.742,A -85,B 0,C 180,E1 19888.315,E2 19888.315} C_VEL
LIN {X 0,Y 407.913,Z 1138.104,A -85,B 0,C 180,E1 19885.079,E2 19885.079} C_VEL
LIN {X 0,Y 407.958,Z 1135.531,A -85,B 0,C 180,E1 19882.395,E2 19882.395} C_VEL
LIN {X 0,Y 408.175,Z 1131.051,A -85,B 0,C 180,E1 19879.199,E2 19879.199} C_VEL
LIN {X 0,Y 408.599,Z 1125.277,A -85,B 0,C 180,E1 19876.125,E2 19876.125} C_VEL
LIN {X 0,Y 409.447,Z 1117.423,A -85,B 0,C 180,E1 19872.814,E2 19872.814} C_VEL
LIN {X 0,Y 410.608,Z 1108.993,A -85,B 0,C 180,E1 19869.919,E2 19869.919} C_VEL
LIN {X 0,Y 412.454,Z 1097.828,A -85,B 0,C 180,E1 19866.725,E2 19866.725} C_VEL
LIN {X 0,Y 414.746,Z 1085.866,A -85,B 0,C 180,E1 19863.822,E2 19863.822} C_VEL
LIN {X 0,Y 417.478,Z 1072.405,A -85,B 0,C 180,E1 19861.067,E2 19861.067} C_VEL
LIN {X 0,Y 420.65,Z 1057.777,A -85,B 0,C 180,E1 19858.471,E2 19858.471} C_VEL
LIN {X 0,Y 424.095,Z 1042.017,A -85,B 0,C 180,E1 19856.087,E2 19856.087} C_VEL
LIN {X 0,Y 428.142,Z 1023.441,A -85,B 0,C 180,E1 19853.677,E2 19853.677} C_VEL
LIN {X 0,Y 431.72,Z 1006.553,A -85,B 0,C 180,E1 19851.803,E2 19851.803} C_VEL
LIN {X 0,Y 435.55,Z 987.488,A -85,B 0,C 180,E1 19850.001,E2 19850.001} C_VEL
LIN {X 0,Y 438.914,Z 969.448,A -85,B 0,C 180,E1 19848.545,E2 19848.545} C_VEL
LIN {X 0,Y 442.498,Z 947.92,A -85,B 0,C 180,E1 19847.091,E2 19847.091} C_VEL
LIN {X 0,Y 445.407,Z 928.173,A -85,B 0,C 180,E1 19845.991,E2 19845.991} C_VEL
LIN {X 0,Y 448.164,Z 905.373,A -85,B 0,C 180,E1 19844.979,E2 19844.979} C_VEL
LIN {X 0,Y 450.42,Z 882.522,A -85,B 0,C 180,E1 19844.203,E2 19844.203} C_VEL
LIN {X 0,Y 451.904,Z 859.641,A -85,B 0,C 180,E1 19843.664,E2 19843.664} C_VEL
LIN {X 0,Y 459.159,Z 661.153,A -85,B 0,C 180,E1 19840.049,E2 19840.049} C_VEL
LIN {X 0,Y 461.377,Z 600.298,A -85,B 0,C 180,E1 19838.917,E2 19838.917} C_VEL
LIN {X 0,Y 450.99,Z 585.376,A -85,B 0,C 180,E1 19836.849,E2 19836.849} C_VEL
LIN {X 0,Y 443.641,Z 575.384,A -85,B 0,C 180,E1 19835.277,E2 19835.277} C_VEL
LIN {X 0,Y 436.321,Z 565.803,A -85,B 0,C 180,E1 19833.602,E2 19833.602} C_VEL
LIN {X 0,Y 432.598,Z 561.061,A -85,B 0,C 180,E1 19832.702,E2 19832.702} C_VEL
LIN {X 0,Y 428.386,Z 555.791,A -85,B 0,C 180,E1 19831.64,E2 19831.64} C_VEL
LIN {X 0,Y 424.976,Z 551.534,A -85,B 0,C 180,E1 19830.74,E2 19830.74} C_VEL
LIN {X 0,Y 423.74,Z 550.094,A -85,B 0,C 180,E1 19830.407,E2 19830.407} C_VEL
LIN {X 0,Y 420.519,Z 546.326,A -85,B 0,C 180,E1 19829.515,E2 19829.515} C_VEL
LIN {X 0,Y 419.394,Z 544.593,A -85,B 0,C 180,E1 19829.179,E2 19829.179} C_VEL
LIN {X 0,Y 416.252,Z 541.66,A -85,B 0,C 180,E1 19828.282,E2 19828.282} C_VEL
LIN {X 0,Y 414.387,Z 538.475,A -85,B 0,C 180,E1 19827.677,E2 19827.677} C_VEL
LIN {X 0,Y 411.335,Z 536.299,A -85,B 0,C 180,E1 19826.763,E2 19826.763} C_VEL
LIN {X 0,Y 409.723,Z 533.468,A -85,B 0,C 180,E1 19826.197,E2 19826.197} C_VEL
LIN {X 0,Y 409.404,Z 532.043,A -85,B 0,C 180,E1 19826.007,E2 19826.007} C_VEL
LIN {X 0,Y 409.435,Z 532.001,A -85,B 0,C 180,E1 19822.242,E2 19822.242} C_VEL
LIN {X 0,Y 409.438,Z 531.999,A -85,B 0,C 180,E1 19818.362,E2 19818.362} C_VEL
LIN {X 0,Y 409.438,Z 532.037,A -85,B 0,C 180,E1 19814.424,E2 19814.424} C_VEL
LIN {X 0,Y 409.42,Z 532.046,A -85,B 0,C 180,E1 19810.554,E2 19810.554} C_VEL
LIN {X 0,Y 409.417,Z 532.049,A -85,B 0,C 180,E1 19806.732,E2 19806.732} C_VEL
LIN {X 0,Y 409.423,Z 532.049,A -85,B 0,C 180,E1 19802.775,E2 19802.775} C_VEL
LIN {X 0,Y 409.439,Z 532.045,A -85,B 0,C 180,E1 19798.881,E2 19798.881} C_VEL
LIN {X 0,Y 409.437,Z 532.041,A -85,B 0,C 180,E1 19794.957,E2 19794.957} C_VEL
LIN {X 0,Y 409.429,Z 532.027,A -85,B 0,C 180,E1 19791.009,E2 19791.009} C_VEL
LIN {X 0,Y 409.425,Z 532.011,A -85,B 0,C 180,E1 19787.008,E2 19787.008} C_VEL
LIN {X 0,Y 409.43,Z 531.999,A -85,B 0,C 180,E1 19783.195,E2 19783.195} C_VEL
LIN {X 0,Y 409.444,Z 532.049,A -85,B 0,C 180,E1 19779.263,E2 19779.263} C_VEL
LIN {X 0,Y 409.438,Z 532.003,A -85,B 0,C 180,E1 19775.29,E2 19775.29} C_VEL
LIN {X 0,Y 409.456,Z 532.229,A -85,B 0,C 180,E1 19774.747,E2 19774.747} C_VEL
LIN {X 0,Y 410.786,Z 535.613,A -85,B 0,C 180,E1 19773.9,E2 19773.9} C_VEL
LIN {X 0,Y 413.727,Z 538.602,A -85,B 0,C 180,E1 19772.978,E2 19772.978} C_VEL
LIN {X 0,Y 416.58,Z 542.284,A -85,B 0,C 180,E1 19772.094,E2 19772.094} C_VEL
LIN {X 0,Y 418.277,Z 544.178,A -85,B 0,C 180,E1 19771.596,E2 19771.596} C_VEL
LIN {X 0,Y 421.695,Z 548.626,A -85,B 0,C 180,E1 19770.607,E2 19770.607} C_VEL
LIN {X 0,Y 423.875,Z 551.582,A -85,B 0,C 180,E1 19769.995,E2 19769.995} C_VEL
LIN {X 0,Y 430.59,Z 560.214,A -85,B 0,C 180,E1 19768.229,E2 19768.229} C_VEL
LIN {X 0,Y 438.931,Z 571.828,A -85,B 0,C 180,E1 19766.194,E2 19766.194} C_VEL
LIN {X 0,Y 447.83,Z 584.661,A -85,B 0,C 180,E1 19764.2,E2 19764.2} C_VEL
LIN {X 0,Y 458.64,Z 601.458,A -85,B 0,C 180,E1 19761.966,E2 19761.966} C_VEL
LIN {X 0,Y 461.612,Z 606.613,A -85,B 0,C 180,E1 19761.376,E2 19761.376} C_VEL
LIN {X 0,Y 453.675,Z 824.139,A -85,B 0,C 180,E1 19757.411,E2 19757.411} C_VEL
LIN {X 0,Y 451.151,Z 891.02,A -85,B 0,C 180,E1 19756.178,E2 19756.178} C_VEL
LIN {X 0,Y 449.174,Z 914.266,A -85,B 0,C 180,E1 19755.56,E2 19755.56} C_VEL
LIN {X 0,Y 446.741,Z 936.931,A -85,B 0,C 180,E1 19754.74,E2 19754.74} C_VEL
LIN {X 0,Y 443.921,Z 957.993,A -85,B 0,C 180,E1 19753.746,E2 19753.746} C_VEL
LIN {X 0,Y 440.595,Z 979.82,A -85,B 0,C 180,E1 19752.479,E2 19752.479} C_VEL
LIN {X 0,Y 437.218,Z 999.291,A -85,B 0,C 180,E1 19751.107,E2 19751.107} C_VEL
LIN {X 0,Y 433.212,Z 1020.615,A -85,B 0,C 180,E1 19749.321,E2 19749.321} C_VEL
LIN {X 0,Y 429.679,Z 1038.373,A -85,B 0,C 180,E1 19747.566,E2 19747.566} C_VEL
LIN {X 0,Y 425.775,Z 1057.365,A -85,B 0,C 180,E1 19745.371,E2 19745.371} C_VEL
LIN {X 0,Y 422.331,Z 1073.925,A -85,B 0,C 180,E1 19743.154,E2 19743.154} C_VEL
LIN {X 0,Y 419.09,Z 1089.657,A -85,B 0,C 180,E1 19740.701,E2 19740.701} C_VEL
LIN {X 0,Y 416.216,Z 1104.282,A -85,B 0,C 180,E1 19738.089,E2 19738.089} C_VEL
LIN {X 0,Y 413.751,Z 1117.476,A -85,B 0,C 180,E1 19735.324,E2 19735.324} C_VEL
LIN {X 0,Y 411.76,Z 1129.547,A -85,B 0,C 180,E1 19732.41,E2 19732.41} C_VEL
LIN {X 0,Y 410.214,Z 1140.127,A -85,B 0,C 180,E1 19729.359,E2 19729.359} C_VEL
LIN {X 0,Y 409.123,Z 1149.409,A -85,B 0,C 180,E1 19726.168,E2 19726.168} C_VEL
LIN {X 0,Y 408.49,Z 1156.181,A -85,B 0,C 180,E1 19723.302,E2 19723.302} C_VEL
LIN {X 0,Y 408.118,Z 1161.81,A -85,B 0,C 180,E1 19720.302,E2 19720.302} C_VEL
LIN {X 0,Y 407.944,Z 1165.799,A -85,B 0,C 180,E1 19717.322,E2 19717.322} C_VEL
LIN {X 0,Y 407.913,Z 1168.523,A -85,B 0,C 180,E1 19714.358,E2 19714.358} C_VEL
LIN {X 0,Y 407.904,Z 1169.803,A -85,B 0,C 180,E1 19711.264,E2 19711.264} C_VEL
LIN {X 0,Y 407.907,Z 1169.78,A -85,B 0,C 180,E1 19708.595,E2 19708.595} C_VEL
LIN {X 0,Y 407.912,Z 1168.294,A -85,B 0,C 180,E1 19705.36,E2 19705.36} C_VEL
LIN {X 0,Y 407.953,Z 1165.638,A -85,B 0,C 180,E1 19702.536,E2 19702.536} C_VEL
LIN {X 0,Y 408.155,Z 1161.352,A -85,B 0,C 180,E1 19699.413,E2 19699.413} C_VEL
LIN {X 0,Y 408.515,Z 1155.867,A -85,B 0,C 180,E1 19696.554,E2 19696.554} C_VEL
LIN {X 0,Y 409.205,Z 1148.66,A -85,B 0,C 180,E1 19693.534,E2 19693.534} C_VEL
LIN {X 0,Y 410.27,Z 1139.658,A -85,B 0,C 180,E1 19690.495,E2 19690.495} C_VEL
LIN {X 0,Y 411.845,Z 1129.002,A -85,B 0,C 180,E1 19687.444,E2 19687.444} C_VEL
LIN {X 0,Y 413.866,Z 1116.828,A -85,B 0,C 180,E1 19684.53,E2 19684.53} C_VEL
LIN {X 0,Y 416.503,Z 1102.71,A -85,B 0,C 180,E1 19681.619,E2 19681.619} C_VEL
LIN {X 0,Y 419.274,Z 1088.761,A -85,B 0,C 180,E1 19679.148,E2 19679.148} C_VEL
LIN {X 0,Y 422.896,Z 1071.148,A -85,B 0,C 180,E1 19676.458,E2 19676.458} C_VEL
LIN {X 0,Y 426.507,Z 1053.997,A -85,B 0,C 180,E1 19674.205,E2 19674.205} C_VEL
LIN {X 0,Y 430.285,Z 1035.288,A -85,B 0,C 180,E1 19672.113,E2 19672.113} C_VEL
LIN {X 0,Y 434.266,Z 1015.316,A -85,B 0,C 180,E1 19670.202,E2 19670.202} C_VEL
LIN {X 0,Y 437.705,Z 996.546,A -85,B 0,C 180,E1 19668.687,E2 19668.687} C_VEL
LIN {X 0,Y 441.328,Z 975.154,A -85,B 0,C 180,E1 19667.226,E2 19667.226} C_VEL
LIN {X 0,Y 444.387,Z 954.584,A -85,B 0,C 180,E1 19666.078,E2 19666.078} C_VEL
LIN {X 0,Y 447.465,Z 930.585,A -85,B 0,C 180,E1 19665.013,E2 19665.013} C_VEL
LIN {X 0,Y 449.643,Z 909.606,A -85,B 0,C 180,E1 19664.301,E2 19664.301} C_VEL
LIN {X 0,Y 451.411,Z 885.556,A -85,B 0,C 180,E1 19663.714,E2 19663.714} C_VEL
LIN {X 0,Y 458.223,Z 696.048,A -85,B 0,C 180,E1 19660.263,E2 19660.263} C_VEL
LIN {X 0,Y 461.515,Z 606.116,A -85,B 0,C 180,E1 19658.604,E2 19658.604} C_VEL
LIN {X 0,Y 449.726,Z 587.502,A -85,B 0,C 180,E1 19656.216,E2 19656.216} C_VEL
LIN {X 0,Y 439.866,Z 573.173,A -85,B 0,C 180,E1 19654.038,E2 19654.038} C_VEL
LIN {X 0,Y 432.629,Z 563.132,A -85,B 0,C 180,E1 19652.306,E2 19652.306} C_VEL
LIN {X 0,Y 425.83,Z 554.019,A -85,B 0,C 180,E1 19650.553,E2 19650.553} C_VEL
LIN {X 0,Y 421.736,Z 548.67,A -85,B 0,C 180,E1 19649.429,E2 19649.429} C_VEL
LIN {X 0,Y 418.407,Z 544.423,A -85,B 0,C 180,E1 19648.472,E2 19648.472} C_VEL
LIN {X 0,Y 416.932,Z 542.605,A -85,B 0,C 180,E1 19648.036,E2 19648.036} C_VEL
LIN {X 0,Y 413.84,Z 538.827,A -85,B 0,C 180,E1 19647.092,E2 19647.092} C_VEL
LIN {X 0,Y 412.828,Z 537.628,A -85,B 0,C 180,E1 19646.774,E2 19646.774} C_VEL
LIN {X 0,Y 410.42,Z 535.033,A -85,B 0,C 180,E1 19646.009,E2 19646.009} C_VEL
LIN {X 0,Y 409.425,Z 532.006,A -85,B 0,C 180,E1 19645.199,E2 19645.199} C_VEL
LIN {X 0,Y 409.419,Z 532.032,A -85,B 0,C 180,E1 19641.338,E2 19641.338} C_VEL
LIN {X 0,Y 409.415,Z 531.988,A -85,B 0,C 180,E1 19637.48,E2 19637.48} C_VEL
LIN {X 0,Y 409.434,Z 532.04,A -85,B 0,C 180,E1 19633.558,E2 19633.558} C_VEL
LIN {X 0,Y 409.432,Z 531.998,A -85,B 0,C 180,E1 19629.558,E2 19629.558} C_VEL
LIN {X 0,Y 409.43,Z 532.033,A -85,B 0,C 180,E1 19625.746,E2 19625.746} C_VEL
LIN {X 0,Y 409.429,Z 532.034,A -85,B 0,C 180,E1 19621.819,E2 19621.819} C_VEL
LIN {X 0,Y 409.436,Z 532.033,A -85,B 0,C 180,E1 19618.04,E2 19618.04} C_VEL
LIN {X 0,Y 409.44,Z 532.034,A -85,B 0,C 180,E1 19614.113,E2 19614.113} C_VEL
LIN {X 0,Y 409.434,Z 531.989,A -85,B 0,C 180,E1 19610.157,E2 19610.157} C_VEL
LIN {X 0,Y 409.444,Z 532.045,A -85,B 0,C 180,E1 19606.154,E2 19606.154} C_VEL
LIN {X 0,Y 409.417,Z 531.989,A -85,B 0,C 180,E1 19602.225,E2 19602.225} C_VEL
LIN {X 0,Y 409.405,Z 532.031,A -85,B 0,C 180,E1 19598.36,E2 19598.36} C_VEL
LIN {X 0,Y 409.397,Z 532.019,A -85,B 0,C 180,E1 19594.387,E2 19594.387} C_VEL
LIN {X 0,Y 409.443,Z 532.232,A -85,B 0,C 180,E1 19593.807,E2 19593.807} C_VEL
LIN {X 0,Y 410.451,Z 535.06,A -85,B 0,C 180,E1 19593.409,E2 19593.409} C_VEL
LIN {X 0,Y 412.966,Z 537.747,A -85,B 0,C 180,E1 19592.611,E2 19592.611} C_VEL
LIN {X 0,Y 414.734,Z 538.914,A -85,B 0,C 180,E1 19592.095,E2 19592.095} C_VEL
LIN {X 0,Y 416.977,Z 542.573,A -85,B 0,C 180,E1 19591.381,E2 19591.381} C_VEL
LIN {X 0,Y 419.932,Z 545.277,A -85,B 0,C 180,E1 19590.549,E2 19590.549} C_VEL
LIN {X 0,Y 422.952,Z 549.383,A -85,B 0,C 180,E1 19589.687,E2 19589.687} C_VEL
LIN {X 0,Y 424.883,Z 551.381,A -85,B 0,C 180,E1 19589.175,E2 19589.175} C_VEL
LIN {X 0,Y 428.291,Z 555.7,A -85,B 0,C 180,E1 19588.274,E2 19588.274} C_VEL
LIN {X 0,Y 430.033,Z 557.868,A -85,B 0,C 180,E1 19587.829,E2 19587.829} C_VEL
LIN {X 0,Y 434.666,Z 563.668,A -85,B 0,C 180,E1 19586.688,E2 19586.688} C_VEL
LIN {X 0,Y 442.433,Z 573.731,A -85,B 0,C 180,E1 19584.89,E2 19584.89} C_VEL
LIN {X 0,Y 452.711,Z 587.674,A -85,B 0,C 180,E1 19582.7,E2 19582.7} C_VEL
LIN {X 0,Y 461.454,Z 600.612,A -85,B 0,C 180,E1 19580.967,E2 19580.967} C_VEL
LIN {X 0,Y 453.748,Z 809.265,A -85,B 0,C 180,E1 19577.165,E2 19577.165} C_VEL
LIN {X 0,Y 451.464,Z 868.113,A -85,B 0,C 180,E1 19576.073,E2 19576.073} C_VEL
LIN {X 0,Y 449.657,Z 890.579,A -85,B 0,C 180,E1 19575.453,E2 19575.453} C_VEL
LIN {X 0,Y 447.347,Z 913.045,A -85,B 0,C 180,E1 19574.619,E2 19574.619} C_VEL
LIN {X 0,Y 444.692,Z 933.217,A -85,B 0,C 180,E1 19573.652,E2 19573.652} C_VEL
LIN {X 0,Y 441.573,Z 953.973,A -85,B 0,C 180,E1 19572.443,E2 19572.443} C_VEL
LIN {X 0,Y 439.612,Z 960.947,A -85,B 0,C 180,E1 19572.065,E2 19572.065} C_VEL
LIN {X 0,Y 431.913,Z 978.625,A -85,B 0,C 180,E1 19571.299,E2 19571.299} C_VEL
LIN {X 0,Y 429.854,Z 985.144,A -85,B 0,C 180,E1 19570.836,E2 19570.836} C_VEL
LIN {X 0,Y 425.884,Z 1004.426,A -85,B 0,C 180,E1 19569.042,E2 19569.042} C_VEL
LIN {X 0,Y 421.783,Z 1022.657,A -85,B 0,C 180,E1 19567.023,E2 19567.023} C_VEL
LIN {X 0,Y 417.732,Z 1040.426,A -85,B 0,C 180,E1 19564.727,E2 19564.727} C_VEL
LIN {X 0,Y 414.141,Z 1055.753,A -85,B 0,C 180,E1 19562.411,E2 19562.411} C_VEL
LIN {X 0,Y 410.475,Z 1071.753,A -85,B 0,C 180,E1 19559.587,E2 19559.587} C_VEL
LIN {X 0,Y 407.549,Z 1085.122,A -85,B 0,C 180,E1 19556.835,E2 19556.835} C_VEL
LIN {X 0,Y 405.051,Z 1097.248,A -85,B 0,C 180,E1 19553.881,E2 19553.881} C_VEL
LIN {X 0,Y 403.1,Z 1108.139,A -85,B 0,C 180,E1 19550.776,E2 19550.776} C_VEL
LIN {X 0,Y 401.704,Z 1117.092,A -85,B 0,C 180,E1 19547.678,E2 19547.678} C_VEL
LIN {X 0,Y 400.732,Z 1125.104,A -85,B 0,C 180,E1 19544.301,E2 19544.301} C_VEL
LIN {X 0,Y 400.269,Z 1130.561,A -85,B 0,C 180,E1 19541.382,E2 19541.382} C_VEL
LIN {X 0,Y 400.001,Z 1135.43,A -85,B 0,C 180,E1 19537.902,E2 19537.902} C_VEL
LIN {X 0,Y 399.919,Z 1138.11,A -85,B 0,C 180,E1 19535.02,E2 19535.02} C_VEL
LIN {X 0,Y 399.903,Z 1139.755,A -85,B 0,C 180,E1 19531.72,E2 19531.72} C_VEL
LIN {X 0,Y 399.894,Z 1139.856,A -85,B 0,C 180,E1 19528.854,E2 19528.854} C_VEL
LIN {X 0,Y 399.912,Z 1138.792,A -85,B 0,C 180,E1 19525.842,E2 19525.842} C_VEL
LIN {X 0,Y 399.947,Z 1136.149,A -85,B 0,C 180,E1 19522.675,E2 19522.675} C_VEL
LIN {X 0,Y 400.107,Z 1132.736,A -85,B 0,C 180,E1 19519.926,E2 19519.926} C_VEL
LIN {X 0,Y 400.549,Z 1127.056,A -85,B 0,C 180,E1 19516.577,E2 19516.577} C_VEL
LIN {X 0,Y 401.264,Z 1120.575,A -85,B 0,C 180,E1 19513.604,E2 19513.604} C_VEL
LIN {X 0,Y 402.534,Z 1111.539,A -85,B 0,C 180,E1 19510.257,E2 19510.257} C_VEL
LIN {X 0,Y 404.191,Z 1101.951,A -85,B 0,C 180,E1 19507.3,E2 19507.3} C_VEL
LIN {X 0,Y 406.395,Z 1090.527,A -85,B 0,C 180,E1 19504.341,E2 19504.341} C_VEL
LIN {X 0,Y 409.113,Z 1077.957,A -85,B 0,C 180,E1 19501.538,E2 19501.538} C_VEL
LIN {X 0,Y 412.248,Z 1063.947,A -85,B 0,C 180,E1 19498.888,E2 19498.888} C_VEL
LIN {X 0,Y 415.865,Z 1048.463,A -85,B 0,C 180,E1 19496.345,E2 19496.345} C_VEL
LIN {X 0,Y 419.556,Z 1032.447,A -85,B 0,C 180,E1 19494.109,E2 19494.109} C_VEL
LIN {X 0,Y 423.738,Z 1014.111,A -85,B 0,C 180,E1 19491.9,E2 19491.9} C_VEL
LIN {X 0,Y 427.526,Z 996.48,A -85,B 0,C 180,E1 19490.094,E2 19490.094} C_VEL
LIN {X 0,Y 431.785,Z 975.309,A -85,B 0,C 180,E1 19488.26,E2 19488.26} C_VEL
LIN {X 0,Y 435.236,Z 956.488,A -85,B 0,C 180,E1 19486.896,E2 19486.896} C_VEL
LIN {X 0,Y 438.714,Z 934.845,A -85,B 0,C 180,E1 19485.599,E2 19485.599} C_VEL
LIN {X 0,Y 441.375,Z 915.599,A -85,B 0,C 180,E1 19484.658,E2 19484.658} C_VEL
LIN {X 0,Y 443.974,Z 892.148,A -85,B 0,C 180,E1 19483.759,E2 19483.759} C_VEL
LIN {X 0,Y 445.768,Z 871.094,A -85,B 0,C 180,E1 19483.162,E2 19483.162} C_VEL
LIN {X 0,Y 447.332,Z 837.532,A -85,B 0,C 180,E1 19482.502,E2 19482.502} C_VEL
LIN {X 0,Y 455.567,Z 624.482,A -85,B 0,C 180,E1 19478.601,E2 19478.601} C_VEL
LIN {X 0,Y 456.259,Z 604.364,A -85,B 0,C 180,E1 19478.209,E2 19478.209} C_VEL
LIN {X 0,Y 444.594,Z 587.528,A -85,B 0,C 180,E1 19475.783,E2 19475.783} C_VEL
LIN {X 0,Y 433.915,Z 573.246,A -85,B 0,C 180,E1 19473.338,E2 19473.338} C_VEL
LIN {X 0,Y 429.273,Z 567.427,A -85,B 0,C 180,E1 19472.195,E2 19472.195} C_VEL
LIN {X 0,Y 425.356,Z 562.482,A -85,B 0,C 180,E1 19471.18,E2 19471.18} C_VEL
LIN {X 0,Y 421.117,Z 557.159,A -85,B 0,C 180,E1 19470.026,E2 19470.026} C_VEL
LIN {X 0,Y 417.655,Z 552.931,A -85,B 0,C 180,E1 19469.038,E2 19469.038} C_VEL
LIN {X 0,Y 416.488,Z 551.529,A -85,B 0,C 180,E1 19468.695,E2 19468.695} C_VEL
LIN {X 0,Y 413.24,Z 547.957,A -85,B 0,C 180,E1 19467.721,E2 19467.721} C_VEL
LIN {X 0,Y 411.764,Z 545.759,A -85,B 0,C 180,E1 19467.24,E2 19467.24} C_VEL
LIN {X 0,Y 408.613,Z 542.956,A -85,B 0,C 180,E1 19466.25,E2 19466.25} C_VEL
LIN {X 0,Y 406.713,Z 539.566,A -85,B 0,C 180,E1 19465.56,E2 19465.56} C_VEL
LIN {X 0,Y 403.592,Z 537.465,A -85,B 0,C 180,E1 19464.517,E2 19464.517} C_VEL
LIN {X 0,Y 401.834,Z 534.605,A -85,B 0,C 180,E1 19463.83,E2 19463.83} C_VEL
LIN {X 0,Y 401.452,Z 532.982,A -85,B 0,C 180,E1 19463.605,E2 19463.605} C_VEL
LIN {X 0,Y 401.472,Z 533.028,A -85,B 0,C 180,E1 19459.712,E2 19459.712} C_VEL
LIN {X 0,Y 401.493,Z 532.982,A -85,B 0,C 180,E1 19455.899,E2 19455.899} C_VEL
LIN {X 0,Y 401.503,Z 533.021,A -85,B 0,C 180,E1 19452.075,E2 19452.075} C_VEL
LIN {X 0,Y 401.499,Z 533.021,A -85,B 0,C 180,E1 19448.161,E2 19448.161} C_VEL
LIN {X 0,Y 401.486,Z 533.023,A -85,B 0,C 180,E1 19444.285,E2 19444.285} C_VEL
LIN {X 0,Y 401.485,Z 533.025,A -85,B 0,C 180,E1 19440.286,E2 19440.286} C_VEL
LIN {X 0,Y 401.49,Z 533.031,A -85,B 0,C 180,E1 19436.288,E2 19436.288} C_VEL
LIN {X 0,Y 401.496,Z 533.035,A -85,B 0,C 180,E1 19432.272,E2 19432.272} C_VEL
LIN {X 0,Y 401.492,Z 532.975,A -85,B 0,C 180,E1 19428.363,E2 19428.363} C_VEL
LIN {X 0,Y 401.492,Z 533.014,A -85,B 0,C 180,E1 19424.398,E2 19424.398} C_VEL
LIN {X 0,Y 401.483,Z 533.008,A -85,B 0,C 180,E1 19420.355,E2 19420.355} C_VEL
LIN {X 0,Y 401.515,Z 533.158,A -85,B 0,C 180,E1 19416.942,E2 19416.942} C_VEL
LIN {X 0,Y 402.223,Z 535.507,A -85,B 0,C 180,E1 19416.486,E2 19416.486} C_VEL
LIN {X 0,Y 404.376,Z 538.201,A -85,B 0,C 180,E1 19415.69,E2 19415.69} C_VEL
LIN {X 0,Y 406.514,Z 539.8,A -85,B 0,C 180,E1 19414.973,E2 19414.973} C_VEL
LIN {X 0,Y 409.927,Z 544.418,A -85,B 0,C 180,E1 19413.802,E2 19413.802} C_VEL
LIN {X 0,Y 411.534,Z 546.143,A -85,B 0,C 180,E1 19413.291,E2 19413.291} C_VEL
LIN {X 0,Y 415.119,Z 550.323,A -85,B 0,C 180,E1 19412.182,E2 19412.182} C_VEL
LIN {X 0,Y 418.987,Z 555.55,A -85,B 0,C 180,E1 19411.025,E2 19411.025} C_VEL
LIN {X 0,Y 427.757,Z 567.14,A -85,B 0,C 180,E1 19408.624,E2 19408.624} C_VEL
LIN {X 0,Y 438.321,Z 581.94,A -85,B 0,C 180,E1 19406.023,E2 19406.023} C_VEL
LIN {X 0,Y 449.66,Z 599.115,A -85,B 0,C 180,E1 19403.501,E2 19403.501} C_VEL
LIN {X 0,Y 456.464,Z 610.365,A -85,B 0,C 180,E1 19402.091,E2 19402.091} C_VEL
LIN {X 0,Y 448.049,Z 829.8,A -85,B 0,C 180,E1 19398.06,E2 19398.06} C_VEL
LIN {X 0,Y 445.6,Z 891.052,A -85,B 0,C 180,E1 19396.918,E2 19396.918} C_VEL
LIN {X 0,Y 443.523,Z 914.366,A -85,B 0,C 180,E1 19396.292,E2 19396.292} C_VEL
LIN {X 0,Y 440.911,Z 937.378,A -85,B 0,C 180,E1 19395.449,E2 19395.449} C_VEL
LIN {X 0,Y 438.064,Z 957.693,A -85,B 0,C 180,E1 19394.484,E2 19394.484} C_VEL
LIN {X 0,Y 434.413,Z 980.453,A -85,B 0,C 180,E1 19393.146,E2 19393.146} C_VEL
LIN {X 0,Y 431.046,Z 998.986,A -85,B 0,C 180,E1 19391.827,E2 19391.827} C_VEL
LIN {X 0,Y 426.982,Z 1019.64,A -85,B 0,C 180,E1 19390.088,E2 19390.088} C_VEL
LIN {X 0,Y 423.106,Z 1038.063,A -85,B 0,C 180,E1 19388.253,E2 19388.253} C_VEL
LIN {X 0,Y 418.918,Z 1057.369,A -85,B 0,C 180,E1 19385.991,E2 19385.991} C_VEL
LIN {X 0,Y 415.192,Z 1074.316,A -85,B 0,C 180,E1 19383.686,E2 19383.686} C_VEL
LIN {X 0,Y 411.705,Z 1090.202,A -85,B 0,C 180,E1 19381.15,E2 19381.15} C_VEL
LIN {X 0,Y 408.677,Z 1104.72,A -85,B 0,C 180,E1 19378.495,E2 19378.495} C_VEL
LIN {X 0,Y 406.072,Z 1117.809,A -85,B 0,C 180,E1 19375.681,E2 19375.681} C_VEL
LIN {X 0,Y 403.87,Z 1130.287,A -85,B 0,C 180,E1 19372.565,E2 19372.565} C_VEL
LIN {X 0,Y 402.327,Z 1140.285,A -85,B 0,C 180,E1 19369.603,E2 19369.603} C_VEL
LIN {X 0,Y 401.136,Z 1149.805,A -85,B 0,C 180,E1 19366.21,E2 19366.21} C_VEL
LIN {X 0,Y 400.485,Z 1156.496,A -85,B 0,C 180,E1 19363.279,E2 19363.279} C_VEL
LIN {X 0,Y 400.094,Z 1162.238,A -85,B 0,C 180,E1 19360.062,E2 19360.062} C_VEL
LIN {X 0,Y 399.944,Z 1165.852,A -85,B 0,C 180,E1 19357.325,E2 19357.325} C_VEL
LIN {X 0,Y 399.914,Z 1168.605,A -85,B 0,C 180,E1 19354.301,E2 19354.301} C_VEL
LIN {X 0,Y 399.904,Z 1169.802,A -85,B 0,C 180,E1 19351.289,E2 19351.289} C_VEL
LIN {X 0,Y 399.907,Z 1169.779,A -85,B 0,C 180,E1 19348.567,E2 19348.567} C_VEL
LIN {X 0,Y 399.913,Z 1168.257,A -85,B 0,C 180,E1 19345.267,E2 19345.267} C_VEL
LIN {X 0,Y 399.962,Z 1165.522,A -85,B 0,C 180,E1 19342.386,E2 19342.386} C_VEL
LIN {X 0,Y 400.163,Z 1161.362,A -85,B 0,C 180,E1 19339.344,E2 19339.344} C_VEL
LIN {X 0,Y 400.588,Z 1155.249,A -85,B 0,C 180,E1 19336.136,E2 19336.136} C_VEL
LIN {X 0,Y 401.341,Z 1147.979,A -85,B 0,C 180,E1 19333.053,E2 19333.053} C_VEL
LIN {X 0,Y 402.512,Z 1138.877,A -85,B 0,C 180,E1 19329.952,E2 19329.952} C_VEL
LIN {X 0,Y 404.23,Z 1128.103,A -85,B 0,C 180,E1 19326.84,E2 19326.84} C_VEL
LIN {X 0,Y 406.316,Z 1116.514,A -85,B 0,C 180,E1 19324.022,E2 19324.022} C_VEL
LIN {X 0,Y 409.186,Z 1102.171,A -85,B 0,C 180,E1 19321.018,E2 19321.018} C_VEL
LIN {X 0,Y 412.262,Z 1087.62,A -85,B 0,C 180,E1 19318.408,E2 19318.408} C_VEL
LIN {X 0,Y 416.009,Z 1070.522,A -85,B 0,C 180,E1 19315.777,E2 19315.777} C_VEL
LIN {X 0,Y 419.88,Z 1053.101,A -85,B 0,C 180,E1 19313.464,E2 19313.464} C_VEL
LIN {X 0,Y 423.825,Z 1034.666,A -85,B 0,C 180,E1 19311.391,E2 19311.391} C_VEL
LIN {X 0,Y 427.939,Z 1015.002,A -85,B 0,C 180,E1 19309.493,E2 19309.493} C_VEL
LIN {X 0,Y 431.717,Z 995.324,A -85,B 0,C 180,E1 19307.895,E2 19307.895} C_VEL
LIN {X 0,Y 435.616,Z 973.13,A -85,B 0,C 180,E1 19306.39,E2 19306.39} C_VEL
LIN {X 0,Y 438.839,Z 952.467,A -85,B 0,C 180,E1 19305.248,E2 19305.248} C_VEL
LIN {X 0,Y 441.856,Z 929.62,A -85,B 0,C 180,E1 19304.246,E2 19304.246} C_VEL
LIN {X 0,Y 444.11,Z 908.746,A -85,B 0,C 180,E1 19303.54,E2 19303.54} C_VEL
LIN {X 0,Y 445.901,Z 884.935,A -85,B 0,C 180,E1 19302.96,E2 19302.96} C_VEL
LIN {X 0,Y 453.124,Z 694.037,A -85,B 0,C 180,E1 19299.455,E2 19299.455} C_VEL
LIN {X 0,Y 456.353,Z 609.972,A -85,B 0,C 180,E1 19297.89,E2 19297.89} C_VEL
LIN {X 0,Y 445.766,Z 593.157,A -85,B 0,C 180,E1 19295.674,E2 19295.674} C_VEL
LIN {X 0,Y 436.551,Z 579.568,A -85,B 0,C 180,E1 19293.581,E2 19293.581} C_VEL
LIN {X 0,Y 429.186,Z 569.242,A -85,B 0,C 180,E1 19291.769,E2 19291.769} C_VEL
LIN {X 0,Y 422.612,Z 560.388,A -85,B 0,C 180,E1 19290.025,E2 19290.025} C_VEL
LIN {X 0,Y 418.803,Z 555.371,A -85,B 0,C 180,E1 19288.95,E2 19288.95} C_VEL
LIN {X 0,Y 414.504,Z 549.77,A -85,B 0,C 180,E1 19287.667,E2 19287.667} C_VEL
LIN {X 0,Y 411.164,Z 545.556,A -85,B 0,C 180,E1 19286.618,E2 19286.618} C_VEL
LIN {X 0,Y 407.901,Z 541.916,A -85,B 0,C 180,E1 19285.557,E2 19285.557} C_VEL
LIN {X 0,Y 406.045,Z 539.245,A -85,B 0,C 180,E1 19284.902,E2 19284.902} C_VEL
LIN {X 0,Y 403.074,Z 536.873,A -85,B 0,C 180,E1 19283.888,E2 19283.888} C_VEL
LIN {X 0,Y 401.555,Z 533.432,A -85,B 0,C 180,E1 19283.167,E2 19283.167} C_VEL
LIN {X 0,Y 401.492,Z 532.978,A -85,B 0,C 180,E1 19283.015,E2 19283.015} C_VEL
LIN {X 0,Y 401.48,Z 532.995,A -85,B 0,C 180,E1 19279.192,E2 19279.192} C_VEL
LIN {X 0,Y 401.482,Z 533.012,A -85,B 0,C 180,E1 19275.306,E2 19275.306} C_VEL
LIN {X 0,Y 401.489,Z 532.976,A -85,B 0,C 180,E1 19271.492,E2 19271.492} C_VEL
LIN {X 0,Y 401.506,Z 533.035,A -85,B 0,C 180,E1 19267.44,E2 19267.44} C_VEL
LIN {X 0,Y 401.494,Z 533.035,A -85,B 0,C 180,E1 19263.426,E2 19263.426} C_VEL
LIN {X 0,Y 401.488,Z 533.031,A -85,B 0,C 180,E1 19259.429,E2 19259.429} C_VEL
LIN {X 0,Y 401.482,Z 533.025,A -85,B 0,C 180,E1 19255.429,E2 19255.429} C_VEL
LIN {X 0,Y 401.487,Z 533.008,A -85,B 0,C 180,E1 19251.55,E2 19251.55} C_VEL
LIN {X 0,Y 401.493,Z 532.993,A -85,B 0,C 180,E1 19247.633,E2 19247.633} C_VEL
LIN {X 0,Y 401.5,Z 532.985,A -85,B 0,C 180,E1 19243.804,E2 19243.804} C_VEL
LIN {X 0,Y 401.503,Z 533.029,A -85,B 0,C 180,E1 19239.748,E2 19239.748} C_VEL
LIN {X 0,Y 401.494,Z 533.23,A -85,B 0,C 180,E1 19236.207,E2 19236.207} C_VEL
LIN {X 0,Y 402.492,Z 535.994,A -85,B 0,C 180,E1 19235.763,E2 19235.763} C_VEL
LIN {X 0,Y 404.981,Z 538.667,A -85,B 0,C 180,E1 19234.871,E2 19234.871} C_VEL
LIN {X 0,Y 406.965,Z 539.946,A -85,B 0,C 180,E1 19234.223,E2 19234.223} C_VEL
LIN {X 0,Y 409.077,Z 543.542,A -85,B 0,C 180,E1 19233.469,E2 19233.469} C_VEL
LIN {X 0,Y 412.362,Z 546.431,A -85,B 0,C 180,E1 19232.45,E2 19232.45} C_VEL
LIN {X 0,Y 415.293,Z 550.501,A -85,B 0,C 180,E1 19231.529,E2 19231.529} C_VEL
LIN {X 0,Y 417.453,Z 552.59,A -85,B 0,C 180,E1 19230.908,E2 19230.908} C_VEL
LIN {X 0,Y 420.901,Z 556.964,A -85,B 0,C 180,E1 19229.918,E2 19229.918} C_VEL
LIN {X 0,Y 422.551,Z 558.982,A -85,B 0,C 180,E1 19229.463,E2 19229.463} C_VEL
LIN {X 0,Y 427.327,Z 564.939,A -85,B 0,C 180,E1 19228.194,E2 19228.194} C_VEL
LIN {X 0,Y 432.379,Z 571.382,A -85,B 0,C 180,E1 19226.925,E2 19226.925} C_VEL
LIN {X 0,Y 439.462,Z 580.662,A -85,B 0,C 180,E1 19225.254,E2 19225.254} C_VEL
LIN {X 0,Y 449.433,Z 594.372,A -85,B 0,C 180,E1 19223.082,E2 19223.082} C_VEL
LIN {X 0,Y 456.308,Z 604.742,A -85,B 0,C 180,E1 19221.676,E2 19221.676} C_VEL
LIN {X 0,Y 448.211,Z 813.274,A -85,B 0,C 180,E1 19217.847,E2 19217.847} C_VEL
LIN {X 0,Y 445.943,Z 868.555,A -85,B 0,C 180,E1 19216.811,E2 19216.811} C_VEL
LIN {X 0,Y 444.057,Z 891.026,A -85,B 0,C 180,E1 19216.186,E2 19216.186} C_VEL
LIN {X 0,Y 441.66,Z 913.358,A -85,B 0,C 180,E1 19215.351,E2 19215.351} C_VEL
LIN {X 0,Y 438.893,Z 933.529,A -85,B 0,C 180,E1 19214.379,E2 19214.379} C_VEL
LIN {X 0,Y 435.625,Z 954.358,A -85,B 0,C 180,E1 19213.156,E2 19213.156} C_VEL
LIN {X 0,Y 432.129,Z 973.481,A -85,B 0,C 180,E1 19211.789,E2 19211.789} C_VEL
LIN {X 0,Y 429.854,Z 985.144,A -85,B 0,C 180,E1 19210.836,E2 19210.836} C_VEL
LIN {X 0,Y 427.751,Z 991.851,A -85,B 0,C 180,E1 19210.346,E2 19210.346} C_VEL
LIN {X 0,Y 419.457,Z 1008.315,A -85,B 0,C 180,E1 19209.276,E2 19209.276} C_VEL
LIN {X 0,Y 417.31,Z 1014.377,A -85,B 0,C 180,E1 19208.707,E2 19208.707} C_VEL
LIN {X 0,Y 412.985,Z 1032.471,A -85,B 0,C 180,E1 19206.506,E2 19206.506} C_VEL
LIN {X 0,Y 408.91,Z 1049.221,A -85,B 0,C 180,E1 19204.137,E2 19204.137} C_VEL
LIN {X 0,Y 405.088,Z 1064.661,A -85,B 0,C 180,E1 19201.552,E2 19201.552} C_VEL
LIN {X 0,Y 401.602,Z 1079.253,A -85,B 0,C 180,E1 19198.719,E2 19198.719} C_VEL
LIN {X 0,Y 398.893,Z 1091.105,A -85,B 0,C 180,E1 19196.018,E2 19196.018} C_VEL
LIN {X 0,Y 396.334,Z 1103.479,A -85,B 0,C 180,E1 19192.705,E2 19192.705} C_VEL
LIN {X 0,Y 394.625,Z 1112.927,A -85,B 0,C 180,E1 19189.694,E2 19189.694} C_VEL
LIN {X 0,Y 393.332,Z 1121.458,A -85,B 0,C 180,E1 19186.39,E2 19186.39} C_VEL
LIN {X 0,Y 392.561,Z 1128.066,A -85,B 0,C 180,E1 19183.252,E2 19183.252} C_VEL
LIN {X 0,Y 392.125,Z 1133.316,A -85,B 0,C 180,E1 19179.985,E2 19179.985} C_VEL
LIN {X 0,Y 391.956,Z 1136.743,A -85,B 0,C 180,E1 19177.106,E2 19177.106} C_VEL
LIN {X 0,Y 391.914,Z 1139.247,A -85,B 0,C 180,E1 19173.804,E2 19173.804} C_VEL
LIN {X 0,Y 391.897,Z 1140.187,A -85,B 0,C 180,E1 19170.877,E2 19170.877} C_VEL
LIN {X 0,Y 391.917,Z 1139.949,A -85,B 0,C 180,E1 19167.661,E2 19167.661} C_VEL
LIN {X 0,Y 391.929,Z 1138.26,A -85,B 0,C 180,E1 19164.584,E2 19164.584} C_VEL
LIN {X 0,Y 392.043,Z 1135.365,A -85,B 0,C 180,E1 19161.494,E2 19161.494} C_VEL
LIN {X 0,Y 392.322,Z 1130.77,A -85,B 0,C 180,E1 19158.236,E2 19158.236} C_VEL
LIN {X 0,Y 392.888,Z 1125.002,A -85,B 0,C 180,E1 19155.106,E2 19155.106} C_VEL
LIN {X 0,Y 393.923,Z 1117.243,A -85,B 0,C 180,E1 19151.808,E2 19151.808} C_VEL
LIN {X 0,Y 395.45,Z 1108.261,A -85,B 0,C 180,E1 19148.649,E2 19148.649} C_VEL
LIN {X 0,Y 397.565,Z 1097.318,A -85,B 0,C 180,E1 19145.483,E2 19145.483} C_VEL
LIN {X 0,Y 400.243,Z 1085.136,A -85,B 0,C 180,E1 19142.474,E2 19142.474} C_VEL
LIN {X 0,Y 403.248,Z 1072.26,A -85,B 0,C 180,E1 19139.779,E2 19139.779} C_VEL
LIN {X 0,Y 407.08,Z 1056.564,A -85,B 0,C 180,E1 19136.957,E2 19136.957} C_VEL
LIN {X 0,Y 410.849,Z 1041.277,A -85,B 0,C 180,E1 19134.605,E2 19134.605} C_VEL
LIN {X 0,Y 415.111,Z 1023.612,A -85,B 0,C 180,E1 19132.28,E2 19132.28} C_VEL
LIN {X 0,Y 419.309,Z 1005.835,A -85,B 0,C 180,E1 19130.279,E2 19130.279} C_VEL
LIN {X 0,Y 423.52,Z 986.479,A -85,B 0,C 180,E1 19128.441,E2 19128.441} C_VEL
LIN {X 0,Y 427.49,Z 966.979,A -85,B 0,C 180,E1 19126.865,E2 19126.865} C_VEL
LIN {X 0,Y 431.229,Z 945.841,A -85,B 0,C 180,E1 19125.462,E2 19125.462} C_VEL
LIN {X 0,Y 434.648,Z 923.983,A -85,B 0,C 180,E1 19124.275,E2 19124.275} C_VEL
LIN {X 0,Y 437.307,Z 903.143,A -85,B 0,C 180,E1 19123.382,E2 19123.382} C_VEL
LIN {X 0,Y 439.682,Z 879.528,A -85,B 0,C 180,E1 19122.613,E2 19122.613} C_VEL
LIN {X 0,Y 441.122,Z 858.098,A -85,B 0,C 180,E1 19122.117,E2 19122.117} C_VEL
LIN {X 0,Y 449.254,Z 656.267,A -85,B 0,C 180,E1 19118.385,E2 19118.385} C_VEL
LIN {X 0,Y 451.143,Z 608.365,A -85,B 0,C 180,E1 19117.472,E2 19117.472} C_VEL
LIN {X 0,Y 440.076,Z 592.362,A -85,B 0,C 180,E1 19115.087,E2 19115.087} C_VEL
LIN {X 0,Y 430.314,Z 579.268,A -85,B 0,C 180,E1 19112.778,E2 19112.778} C_VEL
LIN {X 0,Y 422.929,Z 569.741,A -85,B 0,C 180,E1 19110.865,E2 19110.865} C_VEL
LIN {X 0,Y 418.071,Z 563.774,A -85,B 0,C 180,E1 19109.516,E2 19109.516} C_VEL
LIN {X 0,Y 414.054,Z 558.724,A -85,B 0,C 180,E1 19108.328,E2 19108.328} C_VEL
LIN {X 0,Y 410.562,Z 554.687,A -85,B 0,C 180,E1 19107.248,E2 19107.248} C_VEL
LIN {X 0,Y 409.387,Z 553.061,A -85,B 0,C 180,E1 19106.862,E2 19106.862} C_VEL
LIN {X 0,Y 406.113,Z 549.844,A -85,B 0,C 180,E1 19105.796,E2 19105.796} C_VEL
LIN {X 0,Y 404.202,Z 546.913,A -85,B 0,C 180,E1 19105.102,E2 19105.102} C_VEL
LIN {X 0,Y 401.007,Z 544.2,A -85,B 0,C 180,E1 19103.98,E2 19103.98} C_VEL
LIN {X 0,Y 399.036,Z 540.605,A -85,B 0,C 180,E1 19103.166,E2 19103.166} C_VEL
LIN {X 0,Y 395.671,Z 538.511,A -85,B 0,C 180,E1 19101.884,E2 19101.884} C_VEL
LIN {X 0,Y 393.936,Z 535.721,A -85,B 0,C 180,E1 19101.1,E2 19101.1} C_VEL
LIN {X 0,Y 393.545,Z 534.017,A -85,B 0,C 180,E1 19100.836,E2 19100.836} C_VEL
LIN {X 0,Y 393.53,Z 533.962,A -85,B 0,C 180,E1 19096.837,E2 19096.837} C_VEL
LIN {X 0,Y 393.533,Z 534.02,A -85,B 0,C 180,E1 19092.92,E2 19092.92} C_VEL
LIN {X 0,Y 393.537,Z 534.015,A -85,B 0,C 180,E1 19088.916,E2 19088.916} C_VEL
LIN {X 0,Y 393.546,Z 534.01,A -85,B 0,C 180,E1 19084.956,E2 19084.956} C_VEL
LIN {X 0,Y 393.561,Z 534.007,A -85,B 0,C 180,E1 19081.019,E2 19081.019} C_VEL
LIN {X 0,Y 393.556,Z 534.009,A -85,B 0,C 180,E1 19077.088,E2 19077.088} C_VEL
LIN {X 0,Y 393.554,Z 534.013,A -85,B 0,C 180,E1 19073.142,E2 19073.142} C_VEL
LIN {X 0,Y 393.547,Z 533.962,A -85,B 0,C 180,E1 19069.164,E2 19069.164} C_VEL
LIN {X 0,Y 393.56,Z 534.024,A -85,B 0,C 180,E1 19065.132,E2 19065.132} C_VEL
LIN {X 0,Y 393.554,Z 533.975,A -85,B 0,C 180,E1 19061.177,E2 19061.177} C_VEL
LIN {X 0,Y 393.581,Z 534.151,A -85,B 0,C 180,E1 19059.598,E2 19059.598} C_VEL
LIN {X 0,Y 394.518,Z 536.94,A -85,B 0,C 180,E1 19059.102,E2 19059.102} C_VEL
LIN {X 0,Y 396.891,Z 539.562,A -85,B 0,C 180,E1 19058.109,E2 19058.109} C_VEL
LIN {X 0,Y 399.228,Z 540.953,A -85,B 0,C 180,E1 19057.236,E2 19057.236} C_VEL
LIN {X 0,Y 401.125,Z 544.365,A -85,B 0,C 180,E1 19056.457,E2 19056.457} C_VEL
LIN {X 0,Y 404.498,Z 547.421,A -85,B 0,C 180,E1 19055.269,E2 19055.269} C_VEL
LIN {X 0,Y 407.787,Z 551.78,A -85,B 0,C 180,E1 19054.123,E2 19054.123} C_VEL
LIN {X 0,Y 409.457,Z 553.763,A -85,B 0,C 180,E1 19053.575,E2 19053.575} C_VEL
LIN {X 0,Y 413.293,Z 558.491,A -85,B 0,C 180,E1 19052.362,E2 19052.362} C_VEL
LIN {X 0,Y 418.426,Z 565.344,A -85,B 0,C 180,E1 19050.826,E2 19050.826} C_VEL
LIN {X 0,Y 425.282,Z 574.563,A -85,B 0,C 180,E1 19048.932,E2 19048.932} C_VEL
LIN {X 0,Y 433.091,Z 585.672,A -85,B 0,C 180,E1 19046.943,E2 19046.943} C_VEL
LIN {X 0,Y 441.642,Z 598.425,A -85,B 0,C 180,E1 19044.937,E2 19044.937} C_VEL
LIN {X 0,Y 451.379,Z 614.016,A -85,B 0,C 180,E1 19042.826,E2 19042.826} C_VEL
LIN {X 0,Y 442.705,Z 829.647,A -85,B 0,C 180,E1 19038.833,E2 19038.833} C_VEL
LIN {X 0,Y 440.142,Z 890.767,A -85,B 0,C 180,E1 19037.683,E2 19037.683} C_VEL
LIN {X 0,Y 437.99,Z 914.075,A -85,B 0,C 180,E1 19037.055,E2 19037.055} C_VEL
LIN {X 0,Y 435.27,Z 937.007,A -85,B 0,C 180,E1 19036.213,E2 19036.213} C_VEL
LIN {X 0,Y 432.283,Z 957.394,A -85,B 0,C 180,E1 19035.242,E2 19035.242} C_VEL
LIN {X 0,Y 428.607,Z 979.385,A -85,B 0,C 180,E1 19033.948,E2 19033.948} C_VEL
LIN {X 0,Y 424.945,Z 998.66,A -85,B 0,C 180,E1 19032.57,E2 19032.57} C_VEL
LIN {X 0,Y 420.686,Z 1019.333,A -85,B 0,C 180,E1 19030.814,E2 19030.814} C_VEL
LIN {X 0,Y 416.606,Z 1037.754,A -85,B 0,C 180,E1 19028.962,E2 19028.962} C_VEL
LIN {X 0,Y 412.218,Z 1056.903,A -85,B 0,C 180,E1 19026.695,E2 19026.695} C_VEL
LIN {X 0,Y 408.337,Z 1073.613,A -85,B 0,C 180,E1 19024.394,E2 19024.394} C_VEL
LIN {X 0,Y 404.531,Z 1089.908,A -85,B 0,C 180,E1 19021.762,E2 19021.762} C_VEL
LIN {X 0,Y 401.245,Z 1104.736,A -85,B 0,C 180,E1 19018.997,E2 19018.997} C_VEL
LIN {X 0,Y 398.536,Z 1117.495,A -85,B 0,C 180,E1 19016.203,E2 19016.203} C_VEL
LIN {X 0,Y 396.168,Z 1129.974,A -85,B 0,C 180,E1 19013.029,E2 19013.029} C_VEL
LIN {X 0,Y 394.574,Z 1139.504,A -85,B 0,C 180,E1 19010.159,E2 19010.159} C_VEL
LIN {X 0,Y 393.315,Z 1148.77,A -85,B 0,C 180,E1 19006.846,E2 19006.846} C_VEL
LIN {X 0,Y 392.588,Z 1155.567,A -85,B 0,C 180,E1 19003.851,E2 19003.851} C_VEL
LIN {X 0,Y 392.131,Z 1161.702,A -85,B 0,C 180,E1 19000.43,E2 19000.43} C_VEL
LIN {X 0,Y 391.964,Z 1165.385,A -85,B 0,C 180,E1 18997.622,E2 18997.622} C_VEL
LIN {X 0,Y 391.915,Z 1168.191,A -85,B 0,C 180,E1 18994.536,E2 18994.536} C_VEL
LIN {X 0,Y 391.909,Z 1169.513,A -85,B 0,C 180,E1 18991.315,E2 18991.315} C_VEL
LIN {X 0,Y 391.912,Z 1169.489,A -85,B 0,C 180,E1 18988.538,E2 18988.538} C_VEL
LIN {X 0,Y 391.917,Z 1167.956,A -85,B 0,C 180,E1 18985.17,E2 18985.17} C_VEL
LIN {X 0,Y 391.977,Z 1165.219,A -85,B 0,C 180,E1 18982.23,E2 18982.23} C_VEL
LIN {X 0,Y 392.189,Z 1161.058,A -85,B 0,C 180,E1 18979.125,E2 18979.125} C_VEL
LIN {X 0,Y 392.639,Z 1154.942,A -85,B 0,C 180,E1 18975.849,E2 18975.849} C_VEL
LIN {X 0,Y 393.451,Z 1147.669,A -85,B 0,C 180,E1 18972.702,E2 18972.702} C_VEL
LIN {X 0,Y 394.719,Z 1138.566,A -85,B 0,C 180,E1 18969.539,E2 18969.539} C_VEL
LIN {X 0,Y 396.562,Z 1127.79,A -85,B 0,C 180,E1 18966.366,E2 18966.366} C_VEL
LIN {X 0,Y 398.931,Z 1115.552,A -85,B 0,C 180,E1 18963.343,E2 18963.343} C_VEL
LIN {X 0,Y 402.132,Z 1100.598,A -85,B 0,C 180,E1 18960.197,E2 18960.197} C_VEL
LIN {X 0,Y 405.585,Z 1085.469,A -85,B 0,C 180,E1 18957.469,E2 18957.469} C_VEL
LIN {X 0,Y 409.346,Z 1069.177,A -85,B 0,C 180,E1 18954.969,E2 18954.969} C_VEL
LIN {X 0,Y 413.465,Z 1051.572,A -85,B 0,C 180,E1 18952.628,E2 18952.628} C_VEL
LIN {X 0,Y 417.523,Z 1033.676,A -85,B 0,C 180,E1 18950.609,E2 18950.609} C_VEL
LIN {X 0,Y 421.78,Z 1014.169,A -85,B 0,C 180,E1 18948.717,E2 18948.717} C_VEL
LIN {X 0,Y 425.727,Z 994.57,A -85,B 0,C 180,E1 18947.118,E2 18947.118} C_VEL
LIN {X 0,Y 429.732,Z 972.817,A -85,B 0,C 180,E1 18945.639,E2 18945.639} C_VEL
LIN {X 0,Y 433.104,Z 952.156,A -85,B 0,C 180,E1 18944.491,E2 18944.491} C_VEL
LIN {X 0,Y 436.234,Z 929.416,A -85,B 0,C 180,E1 18943.489,E2 18943.489} C_VEL
LIN {X 0,Y 438.512,Z 909.194,A -85,B 0,C 180,E1 18942.8,E2 18942.8} C_VEL
LIN {X 0,Y 440.437,Z 884.933,A -85,B 0,C 180,E1 18942.2,E2 18942.2} C_VEL
LIN {X 0,Y 447.975,Z 695.435,A -85,B 0,C 180,E1 18938.691,E2 18938.691} C_VEL
LIN {X 0,Y 451.264,Z 613.874,A -85,B 0,C 180,E1 18937.16,E2 18937.16} C_VEL
LIN {X 0,Y 440.85,Z 597.233,A -85,B 0,C 180,E1 18934.897,E2 18934.897} C_VEL
LIN {X 0,Y 430.779,Z 582.274,A -85,B 0,C 180,E1 18932.501,E2 18932.501} C_VEL
LIN {X 0,Y 420.651,Z 568.172,A -85,B 0,C 180,E1 18929.826,E2 18929.826} C_VEL
LIN {X 0,Y 415.797,Z 561.922,A -85,B 0,C 180,E1 18928.432,E2 18928.432} C_VEL
LIN {X 0,Y 411.885,Z 556.726,A -85,B 0,C 180,E1 18927.231,E2 18927.231} C_VEL
LIN {X 0,Y 407.897,Z 551.881,A -85,B 0,C 180,E1 18925.947,E2 18925.947} C_VEL
LIN {X 0,Y 404.315,Z 547.156,A -85,B 0,C 180,E1 18924.704,E2 18924.704} C_VEL
LIN {X 0,Y 400.676,Z 543.772,A -85,B 0,C 180,E1 18923.415,E2 18923.415} C_VEL
LIN {X 0,Y 398.958,Z 540.567,A -85,B 0,C 180,E1 18922.702,E2 18922.702} C_VEL
LIN {X 0,Y 395.754,Z 538.602,A -85,B 0,C 180,E1 18921.489,E2 18921.489} C_VEL
LIN {X 0,Y 393.984,Z 535.762,A -85,B 0,C 180,E1 18920.694,E2 18920.694} C_VEL
LIN {X 0,Y 393.564,Z 534.02,A -85,B 0,C 180,E1 18920.438,E2 18920.438} C_VEL
LIN {X 0,Y 393.555,Z 533.969,A -85,B 0,C 180,E1 18916.379,E2 18916.379} C_VEL
LIN {X 0,Y 393.555,Z 533.979,A -85,B 0,C 180,E1 18912.471,E2 18912.471} C_VEL
LIN {X 0,Y 393.558,Z 533.999,A -85,B 0,C 180,E1 18908.473,E2 18908.473} C_VEL
LIN {X 0,Y 393.555,Z 534.017,A -85,B 0,C 180,E1 18904.517,E2 18904.517} C_VEL
LIN {X 0,Y 393.561,Z 534.023,A -85,B 0,C 180,E1 18900.436,E2 18900.436} C_VEL
LIN {X 0,Y 393.56,Z 534.027,A -85,B 0,C 180,E1 18896.358,E2 18896.358} C_VEL
LIN {X 0,Y 393.566,Z 534.019,A -85,B 0,C 180,E1 18892.408,E2 18892.408} C_VEL
LIN {X 0,Y 393.548,Z 533.964,A -85,B 0,C 180,E1 18888.421,E2 18888.421} C_VEL
LIN {X 0,Y 393.533,Z 533.997,A -85,B 0,C 180,E1 18884.678,E2 18884.678} C_VEL
LIN {X 0,Y 393.527,Z 533.987,A -85,B 0,C 180,E1 18880.713,E2 18880.713} C_VEL
LIN {X 0,Y 393.566,Z 534.23,A -85,B 0,C 180,E1 18878.97,E2 18878.97} C_VEL
LIN {X 0,Y 394.505,Z 536.967,A -85,B 0,C 180,E1 18878.477,E2 18878.477} C_VEL
LIN {X 0,Y 396.897,Z 539.53,A -85,B 0,C 180,E1 18877.485,E2 18877.485} C_VEL
LIN {X 0,Y 399.197,Z 540.909,A -85,B 0,C 180,E1 18876.629,E2 18876.629} C_VEL
LIN {X 0,Y 401.157,Z 544.38,A -85,B 0,C 180,E1 18875.83,E2 18875.83} C_VEL
LIN {X 0,Y 404.272,Z 546.944,A -85,B 0,C 180,E1 18874.746,E2 18874.746} C_VEL
LIN {X 0,Y 407.635,Z 551.648,A -85,B 0,C 180,E1 18873.564,E2 18873.564} C_VEL
LIN {X 0,Y 410.071,Z 553.875,A -85,B 0,C 180,E1 18872.795,E2 18872.795} C_VEL
LIN {X 0,Y 413.299,Z 558.07,A -85,B 0,C 180,E1 18871.773,E2 18871.773} C_VEL
LIN {X 0,Y 415.089,Z 559.985,A -85,B 0,C 180,E1 18871.243,E2 18871.243} C_VEL
LIN {X 0,Y 418.971,Z 564.635,A -85,B 0,C 180,E1 18870.12,E2 18870.12} C_VEL
LIN {X 0,Y 423.294,Z 570.104,A -85,B 0,C 180,E1 18868.928,E2 18868.928} C_VEL
LIN {X 0,Y 432.379,Z 581.971,A -85,B 0,C 180,E1 18866.608,E2 18866.608} C_VEL
LIN {X 0,Y 442.395,Z 595.666,A -85,B 0,C 180,E1 18864.291,E2 18864.291} C_VEL
LIN {X 0,Y 451.238,Z 608.691,A -85,B 0,C 180,E1 18862.405,E2 18862.405} C_VEL
LIN {X 0,Y 442.765,Z 816.646,A -85,B 0,C 180,E1 18858.559,E2 18858.559} C_VEL
LIN {X 0,Y 440.498,Z 868.991,A -85,B 0,C 180,E1 18857.567,E2 18857.567} C_VEL
LIN {X 0,Y 438.519,Z 891.601,A -85,B 0,C 180,E1 18856.933,E2 18856.933} C_VEL
LIN {X 0,Y 435.946,Z 914.405,A -85,B 0,C 180,E1 18856.069,E2 18856.069} C_VEL
LIN {X 0,Y 433.166,Z 933.841,A -85,B 0,C 180,E1 18855.125,E2 18855.125} C_VEL
LIN {X 0,Y 429.757,Z 954.669,A -85,B 0,C 180,E1 18853.894,E2 18853.894} C_VEL
LIN {X 0,Y 426.11,Z 973.792,A -85,B 0,C 180,E1 18852.516,E2 18852.516} C_VEL
LIN {X 0,Y 422.023,Z 993.555,A -85,B 0,C 180,E1 18850.837,E2 18850.837} C_VEL
LIN {X 0,Y 417.774,Z 1012.266,A -85,B 0,C 180,E1 18848.938,E2 18848.938} C_VEL
LIN {X 0,Y 417.31,Z 1014.377,A -85,B 0,C 180,E1 18848.707,E2 18848.707} C_VEL
LIN {X 0,Y 415.143,Z 1020.459,A -85,B 0,C 180,E1 18848.111,E2 18848.111} C_VEL
LIN {X 0,Y 406.499,Z 1035.713,A -85,B 0,C 180,E1 18846.73,E2 18846.73} C_VEL
LIN {X 0,Y 404.234,Z 1041.241,A -85,B 0,C 180,E1 18846.031,E2 18846.031} C_VEL
LIN {X 0,Y 400.299,Z 1056.381,A -85,B 0,C 180,E1 18843.677,E2 18843.677} C_VEL
LIN {X 0,Y 396.212,Z 1072.154,A -85,B 0,C 180,E1 18840.816,E2 18840.816} C_VEL
LIN {X 0,Y 392.917,Z 1085.452,A -85,B 0,C 180,E1 18837.992,E2 18837.992} C_VEL
LIN {X 0,Y 389.999,Z 1097.875,A -85,B 0,C 180,E1 18834.864,E2 18834.864} C_VEL
LIN {X 0,Y 387.738,Z 1108.763,A -85,B 0,C 180,E1 18831.639,E2 18831.639} C_VEL
LIN {X 0,Y 386.103,Z 1117.713,A -85,B 0,C 180,E1 18828.418,E2 18828.418} C_VEL
LIN {X 0,Y 384.946,Z 1125.72,A -85,B 0,C 180,E1 18824.901,E2 18824.901} C_VEL
LIN {X 0,Y 384.374,Z 1131.172,A -85,B 0,C 180,E1 18821.859,E2 18821.859} C_VEL
LIN {X 0,Y 384.051,Z 1135.882,A -85,B 0,C 180,E1 18818.384,E2 18818.384} C_VEL
LIN {X 0,Y 383.935,Z 1138.603,A -85,B 0,C 180,E1 18815.38,E2 18815.38} C_VEL
LIN {X 0,Y 383.92,Z 1140.312,A -85,B 0,C 180,E1 18812.09,E2 18812.09} C_VEL
LIN {X 0,Y 383.902,Z 1140.478,A -85,B 0,C 180,E1 18808.956,E2 18808.956} C_VEL
LIN {X 0,Y 383.925,Z 1139.523,A -85,B 0,C 180,E1 18805.968,E2 18805.968} C_VEL
LIN {X 0,Y 383.979,Z 1136.906,A -85,B 0,C 180,E1 18802.519,E2 18802.519} C_VEL
LIN {X 0,Y 384.17,Z 1133.541,A -85,B 0,C 180,E1 18799.655,E2 18799.655} C_VEL
LIN {X 0,Y 384.696,Z 1127.958,A -85,B 0,C 180,E1 18796.166,E2 18796.166} C_VEL
LIN {X 0,Y 385.505,Z 1121.627,A -85,B 0,C 180,E1 18793.113,E2 18793.113} C_VEL
LIN {X 0,Y 386.982,Z 1112.6,A -85,B 0,C 180,E1 18789.586,E2 18789.586} C_VEL
LIN {X 0,Y 388.876,Z 1103.067,A -85,B 0,C 180,E1 18786.514,E2 18786.514} C_VEL
LIN {X 0,Y 391.536,Z 1091.14,A -85,B 0,C 180,E1 18783.292,E2 18783.292} C_VEL
LIN {X 0,Y 394.704,Z 1078.286,A -85,B 0,C 180,E1 18780.329,E2 18780.329} C_VEL
LIN {X 0,Y 398.419,Z 1063.588,A -85,B 0,C 180,E1 18777.481,E2 18777.481} C_VEL
LIN {X 0,Y 402.669,Z 1047.311,A -85,B 0,C 180,E1 18774.779,E2 18774.779} C_VEL
LIN {X 0,Y 406.684,Z 1031.739,A -85,B 0,C 180,E1 18772.572,E2 18772.572} C_VEL
LIN {X 0,Y 411.405,Z 1012.737,A -85,B 0,C 180,E1 18770.269,E2 18770.269} C_VEL
LIN {X 0,Y 415.722,Z 994.622,A -85,B 0,C 180,E1 18768.409,E2 18768.409} C_VEL
LIN {X 0,Y 419.987,Z 975.012,A -85,B 0,C 180,E1 18766.714,E2 18766.714} C_VEL
LIN {X 0,Y 423.781,Z 955.983,A -85,B 0,C 180,E1 18765.324,E2 18765.324} C_VEL
LIN {X 0,Y 427.445,Z 934.729,A -85,B 0,C 180,E1 18764.048,E2 18764.048} C_VEL
LIN {X 0,Y 430.39,Z 914.984,A -85,B 0,C 180,E1 18763.079,E2 18763.079} C_VEL
LIN {X 0,Y 433.102,Z 891.968,A -85,B 0,C 180,E1 18762.2,E2 18762.2} C_VEL
LIN {X 0,Y 435.168,Z 869.268,A -85,B 0,C 180,E1 18761.562,E2 18761.562} C_VEL
LIN {X 0,Y 437.617,Z 815.104,A -85,B 0,C 180,E1 18760.529,E2 18760.529} C_VEL
LIN {X 0,Y 446.26,Z 612.74,A -85,B 0,C 180,E1 18756.755,E2 18756.755} C_VEL
LIN {X 0,Y 435.753,Z 597.312,A -85,B 0,C 180,E1 18754.405,E2 18754.405} C_VEL
LIN {X 0,Y 424.462,Z 582.113,A -85,B 0,C 180,E1 18751.609,E2 18751.609} C_VEL
LIN {X 0,Y 418.945,Z 575.255,A -85,B 0,C 180,E1 18750.118,E2 18750.118} C_VEL
LIN {X 0,Y 415.506,Z 570.818,A -85,B 0,C 180,E1 18749.127,E2 18749.127} C_VEL
LIN {X 0,Y 411.427,Z 565.719,A -85,B 0,C 180,E1 18747.893,E2 18747.893} C_VEL
LIN {X 0,Y 407.723,Z 561.107,A -85,B 0,C 180,E1 18746.704,E2 18746.704} C_VEL
LIN {X 0,Y 403.458,Z 556.459,A -85,B 0,C 180,E1 18745.27,E2 18745.27} C_VEL
LIN {X 0,Y 402.118,Z 554.379,A -85,B 0,C 180,E1 18744.77,E2 18744.77} C_VEL
LIN {X 0,Y 398.721,Z 551.232,A -85,B 0,C 180,E1 18743.538,E2 18743.538} C_VEL
LIN {X 0,Y 396.897,Z 548.152,A -85,B 0,C 180,E1 18742.776,E2 18742.776} C_VEL
LIN {X 0,Y 393.571,Z 545.705,A -85,B 0,C 180,E1 18741.459,E2 18741.459} C_VEL
LIN {X 0,Y 391.644,Z 542.418,A -85,B 0,C 180,E1 18740.551,E2 18740.551} C_VEL
LIN {X 0,Y 391.212,Z 541.672,A -85,B 0,C 180,E1 18740.34,E2 18740.34} C_VEL
LIN {X 0,Y 387.956,Z 539.721,A -85,B 0,C 180,E1 18738.872,E2 18738.872} C_VEL
LIN {X 0,Y 386.046,Z 536.769,A -85,B 0,C 180,E1 18737.835,E2 18737.835} C_VEL
LIN {X 0,Y 385.584,Z 534.951,A -85,B 0,C 180,E1 18737.467,E2 18737.467} C_VEL
LIN {X 0,Y 385.607,Z 535.016,A -85,B 0,C 180,E1 18733.496,E2 18733.496} C_VEL
LIN {X 0,Y 385.619,Z 535.008,A -85,B 0,C 180,E1 18729.552,E2 18729.552} C_VEL
LIN {X 0,Y 385.622,Z 535.001,A -85,B 0,C 180,E1 18725.505,E2 18725.505} C_VEL
LIN {X 0,Y 385.622,Z 534.997,A -85,B 0,C 180,E1 18721.486,E2 18721.486} C_VEL
LIN {X 0,Y 385.618,Z 534.997,A -85,B 0,C 180,E1 18717.474,E2 18717.474} C_VEL
LIN {X 0,Y 385.621,Z 534.998,A -85,B 0,C 180,E1 18713.449,E2 18713.449} C_VEL
LIN {X 0,Y 385.61,Z 534.95,A -85,B 0,C 180,E1 18709.392,E2 18709.392} C_VEL
LIN {X 0,Y 385.628,Z 535.014,A -85,B 0,C 180,E1 18705.266,E2 18705.266} C_VEL
LIN {X 0,Y 385.63,Z 535.135,A -85,B 0,C 180,E1 18702.944,E2 18702.944} C_VEL
LIN {X 0,Y 386.493,Z 537.752,A -85,B 0,C 180,E1 18702.382,E2 18702.382} C_VEL
LIN {X 0,Y 388.869,Z 540.459,A -85,B 0,C 180,E1 18701.175,E2 18701.175} C_VEL
LIN {X 0,Y 391.486,Z 541.88,A -85,B 0,C 180,E1 18700.022,E2 18700.022} C_VEL
LIN {X 0,Y 393.282,Z 545.354,A -85,B 0,C 180,E1 18699.15,E2 18699.15} C_VEL
LIN {X 0,Y 396.322,Z 547.881,A -85,B 0,C 180,E1 18697.92,E2 18697.92} C_VEL
LIN {X 0,Y 397.193,Z 548.634,A -85,B 0,C 180,E1 18697.582,E2 18697.582} C_VEL
LIN {X 0,Y 399.715,Z 552.426,A -85,B 0,C 180,E1 18696.564,E2 18696.564} C_VEL
LIN {X 0,Y 402.499,Z 554.983,A -85,B 0,C 180,E1 18695.569,E2 18695.569} C_VEL
LIN {X 0,Y 405.876,Z 559.345,A -85,B 0,C 180,E1 18694.377,E2 18694.377} C_VEL
LIN {X 0,Y 410.882,Z 565.692,A -85,B 0,C 180,E1 18692.736,E2 18692.736} C_VEL
LIN {X 0,Y 416.37,Z 573.104,A -85,B 0,C 180,E1 18691.062,E2 18691.062} C_VEL
LIN {X 0,Y 422.934,Z 582.116,A -85,B 0,C 180,E1 18689.215,E2 18689.215} C_VEL
LIN {X 0,Y 432.688,Z 596.151,A -85,B 0,C 180,E1 18686.715,E2 18686.715} C_VEL
LIN {X 0,Y 443.838,Z 613.677,A -85,B 0,C 180,E1 18684.127,E2 18684.127} C_VEL
LIN {X 0,Y 446.372,Z 618.283,A -85,B 0,C 180,E1 18683.562,E2 18683.562} C_VEL
LIN {X 0,Y 437.181,Z 836.002,A -85,B 0,C 180,E1 18679.504,E2 18679.504} C_VEL
LIN {X 0,Y 434.739,Z 890.866,A -85,B 0,C 180,E1 18678.458,E2 18678.458} C_VEL
LIN {X 0,Y 432.508,Z 914.045,A -85,B 0,C 180,E1 18677.828,E2 18677.828} C_VEL
LIN {X 0,Y 429.721,Z 936.598,A -85,B 0,C 180,E1 18676.998,E2 18676.998} C_VEL
LIN {X 0,Y 426.588,Z 957.095,A -85,B 0,C 180,E1 18676.018,E2 18676.018} C_VEL
LIN {X 0,Y 422.742,Z 979.083,A -85,B 0,C 180,E1 18674.72,E2 18674.72} C_VEL
LIN {X 0,Y 418.898,Z 998.434,A -85,B 0,C 180,E1 18673.326,E2 18673.326} C_VEL
LIN {X 0,Y 414.286,Z 1019.769,A -85,B 0,C 180,E1 18671.49,E2 18671.49} C_VEL
LIN {X 0,Y 410.179,Z 1037.446,A -85,B 0,C 180,E1 18669.691,E2 18669.691} C_VEL
LIN {X 0,Y 405.681,Z 1056.02,A -85,B 0,C 180,E1 18667.476,E2 18667.476} C_VEL
LIN {X 0,Y 401.649,Z 1072.473,A -85,B 0,C 180,E1 18665.19,E2 18665.19} C_VEL
LIN {X 0,Y 397.625,Z 1088.713,A -85,B 0,C 180,E1 18662.556,E2 18662.556} C_VEL
LIN {X 0,Y 394.183,Z 1103.338,A -85,B 0,C 180,E1 18659.812,E2 18659.812} C_VEL
LIN {X 0,Y 391.129,Z 1116.719,A -85,B 0,C 180,E1 18656.855,E2 18656.855} C_VEL
LIN {X 0,Y 388.596,Z 1129.134,A -85,B 0,C 180,E1 18653.665,E2 18653.665} C_VEL
LIN {X 0,Y 386.786,Z 1139.192,A -85,B 0,C 180,E1 18650.583,E2 18650.583} C_VEL
LIN {X 0,Y 385.423,Z 1148.461,A -85,B 0,C 180,E1 18647.202,E2 18647.202} C_VEL
LIN {X 0,Y 384.639,Z 1155.26,A -85,B 0,C 180,E1 18644.143,E2 18644.143} C_VEL
LIN {X 0,Y 384.158,Z 1161.398,A -85,B 0,C 180,E1 18640.649,E2 18640.649} C_VEL
LIN {X 0,Y 383.979,Z 1165.083,A -85,B 0,C 180,E1 18637.782,E2 18637.782} C_VEL
LIN {X 0,Y 383.918,Z 1167.89,A -85,B 0,C 180,E1 18634.631,E2 18634.631} C_VEL
LIN {X 0,Y 383.915,Z 1169.213,A -85,B 0,C 180,E1 18631.343,E2 18631.343} C_VEL
LIN {X 0,Y 383.918,Z 1169.189,A -85,B 0,C 180,E1 18628.507,E2 18628.507} C_VEL
LIN {X 0,Y 383.922,Z 1167.655,A -85,B 0,C 180,E1 18625.069,E2 18625.069} C_VEL
LIN {X 0,Y 383.995,Z 1164.917,A -85,B 0,C 180,E1 18622.067,E2 18622.067} C_VEL
LIN {X 0,Y 384.225,Z 1160.5,A -85,B 0,C 180,E1 18618.745,E2 18618.745} C_VEL
LIN {X 0,Y 384.698,Z 1154.635,A -85,B 0,C 180,E1 18615.551,E2 18615.551} C_VEL
LIN {X 0,Y 385.577,Z 1147.36,A -85,B 0,C 180,E1 18612.338,E2 18612.338} C_VEL
LIN {X 0,Y 386.946,Z 1138.254,A -85,B 0,C 180,E1 18609.109,E2 18609.109} C_VEL
LIN {X 0,Y 388.933,Z 1127.464,A -85,B 0,C 180,E1 18605.869,E2 18605.869} C_VEL
LIN {X 0,Y 391.455,Z 1115.237,A -85,B 0,C 180,E1 18602.793,E2 18602.793} C_VEL
LIN {X 0,Y 394.705,Z 1100.981,A -85,B 0,C 180,E1 18599.728,E2 18599.728} C_VEL
LIN {X 0,Y 398.287,Z 1086.129,A -85,B 0,C 180,E1 18596.991,E2 18596.991} C_VEL
LIN {X 0,Y 402.423,Z 1069.219,A -85,B 0,C 180,E1 18594.336,E2 18594.336} C_VEL
LIN {X 0,Y 406.658,Z 1052.169,A -85,B 0,C 180,E1 18592.025,E2 18592.025} C_VEL
LIN {X 0,Y 410.956,Z 1034.114,A -85,B 0,C 180,E1 18589.954,E2 18589.954} C_VEL
LIN {X 0,Y 415.489,Z 1014.373,A -85,B 0,C 180,E1 18588.01,E2 18588.01} C_VEL
LIN {X 0,Y 419.624,Z 994.788,A -85,B 0,C 180,E1 18586.394,E2 18586.394} C_VEL
LIN {X 0,Y 424.034,Z 971.923,A -85,B 0,C 180,E1 18584.832,E2 18584.832} C_VEL
LIN {X 0,Y 427.448,Z 951.845,A -85,B 0,C 180,E1 18583.714,E2 18583.714} C_VEL
LIN {X 0,Y 430.713,Z 929.039,A -85,B 0,C 180,E1 18582.706,E2 18582.706} C_VEL
LIN {X 0,Y 433.051,Z 909.092,A -85,B 0,C 180,E1 18582.023,E2 18582.023} C_VEL
LIN {X 0,Y 435.062,Z 884.776,A -85,B 0,C 180,E1 18581.419,E2 18581.419} C_VEL
LIN {X 0,Y 442.979,Z 695.199,A -85,B 0,C 180,E1 18577.879,E2 18577.879} C_VEL
LIN {X 0,Y 446.214,Z 617.727,A -85,B 0,C 180,E1 18576.407,E2 18576.407} C_VEL
LIN {X 0,Y 436.256,Z 601.735,A -85,B 0,C 180,E1 18574.16,E2 18574.16} C_VEL
LIN {X 0,Y 427.091,Z 588.052,A -85,B 0,C 180,E1 18571.904,E2 18571.904} C_VEL
LIN {X 0,Y 417.812,Z 574.933,A -85,B 0,C 180,E1 18569.378,E2 18569.378} C_VEL
LIN {X 0,Y 412.934,Z 568.56,A -85,B 0,C 180,E1 18567.939,E2 18567.939} C_VEL
LIN {X 0,Y 409.292,Z 563.662,A -85,B 0,C 180,E1 18566.789,E2 18566.789} C_VEL
LIN {X 0,Y 405.371,Z 558.861,A -85,B 0,C 180,E1 18565.493,E2 18565.493} C_VEL
LIN {X 0,Y 401.662,Z 554.059,A -85,B 0,C 180,E1 18564.172,E2 18564.172} C_VEL
LIN {X 0,Y 398.475,Z 550.911,A -85,B 0,C 180,E1 18563.004,E2 18563.004} C_VEL
LIN {X 0,Y 396.933,Z 548.16,A -85,B 0,C 180,E1 18562.356,E2 18562.356} C_VEL
LIN {X 0,Y 393.646,Z 545.793,A -85,B 0,C 180,E1 18561.063,E2 18561.063} C_VEL
LIN {X 0,Y 391.705,Z 542.508,A -85,B 0,C 180,E1 18560.157,E2 18560.157} C_VEL
LIN {X 0,Y 391.443,Z 541.766,A -85,B 0,C 180,E1 18560.015,E2 18560.015} C_VEL
LIN {X 0,Y 388.002,Z 539.724,A -85,B 0,C 180,E1 18558.479,E2 18558.479} C_VEL
LIN {X 0,Y 386.07,Z 536.83,A -85,B 0,C 180,E1 18557.444,E2 18557.444} C_VEL
LIN {X 0,Y 385.603,Z 534.949,A -85,B 0,C 180,E1 18557.076,E2 18557.076} C_VEL
LIN {X 0,Y 385.608,Z 534.987,A -85,B 0,C 180,E1 18553.189,E2 18553.189} C_VEL
LIN {X 0,Y 385.609,Z 534.967,A -85,B 0,C 180,E1 18549.1,E2 18549.1} C_VEL
LIN {X 0,Y 385.619,Z 534.998,A -85,B 0,C 180,E1 18545.206,E2 18545.206} C_VEL
LIN {X 0,Y 385.621,Z 535.002,A -85,B 0,C 180,E1 18541.188,E2 18541.188} C_VEL
LIN {X 0,Y 385.609,Z 535.008,A -85,B 0,C 180,E1 18537.176,E2 18537.176} C_VEL
LIN {X 0,Y 385.605,Z 535.016,A -85,B 0,C 180,E1 18533.149,E2 18533.149} C_VEL
LIN {X 0,Y 385.592,Z 534.947,A -85,B 0,C 180,E1 18529.088,E2 18529.088} C_VEL
LIN {X 0,Y 385.6,Z 534.998,A -85,B 0,C 180,E1 18525.125,E2 18525.125} C_VEL
LIN {X 0,Y 385.613,Z 535.076,A -85,B 0,C 180,E1 18522.304,E2 18522.304} C_VEL
LIN {X 0,Y 386.521,Z 537.773,A -85,B 0,C 180,E1 18521.72,E2 18521.72} C_VEL
LIN {X 0,Y 388.836,Z 540.472,A -85,B 0,C 180,E1 18520.549,E2 18520.549} C_VEL
LIN {X 0,Y 391.456,Z 541.909,A -85,B 0,C 180,E1 18519.4,E2 18519.4} C_VEL
LIN {X 0,Y 393.197,Z 545.251,A -85,B 0,C 180,E1 18518.559,E2 18518.559} C_VEL
LIN {X 0,Y 396.331,Z 547.876,A -85,B 0,C 180,E1 18517.295,E2 18517.295} C_VEL
LIN {X 0,Y 397.201,Z 548.671,A -85,B 0,C 180,E1 18516.956,E2 18516.956} C_VEL
LIN {X 0,Y 399.739,Z 552.44,A -85,B 0,C 180,E1 18515.939,E2 18515.939} C_VEL
LIN {X 0,Y 402.544,Z 554.93,A -85,B 0,C 180,E1 18514.944,E2 18514.944} C_VEL
LIN {X 0,Y 405.51,Z 559.011,A -85,B 0,C 180,E1 18513.888,E2 18513.888} C_VEL
LIN {X 0,Y 407.802,Z 561.249,A -85,B 0,C 180,E1 18513.144,E2 18513.144} C_VEL
LIN {X 0,Y 411.314,Z 565.629,A -85,B 0,C 180,E1 18512.02,E2 18512.02} C_VEL
LIN {X 0,Y 413.585,Z 568.537,A -85,B 0,C 180,E1 18511.322,E2 18511.322} C_VEL
LIN {X 0,Y 417.329,Z 573.105,A -85,B 0,C 180,E1 18510.228,E2 18510.228} C_VEL
LIN {X 0,Y 425.405,Z 583.372,A -85,B 0,C 180,E1 18508.033,E2 18508.033} C_VEL
LIN {X 0,Y 436.655,Z 598.674,A -85,B 0,C 180,E1 18505.278,E2 18505.278} C_VEL
LIN {X 0,Y 446.237,Z 612.794,A -85,B 0,C 180,E1 18503.147,E2 18503.147} C_VEL
LIN {X 0,Y 437.336,Z 821.288,A -85,B 0,C 180,E1 18499.264,E2 18499.264} C_VEL
LIN {X 0,Y 435.122,Z 869.528,A -85,B 0,C 180,E1 18498.339,E2 18498.339} C_VEL
LIN {X 0,Y 433.071,Z 892.047,A -85,B 0,C 180,E1 18497.704,E2 18497.704} C_VEL
LIN {X 0,Y 430.407,Z 914.718,A -85,B 0,C 180,E1 18496.84,E2 18496.84} C_VEL
LIN {X 0,Y 427.406,Z 934.855,A -85,B 0,C 180,E1 18495.853,E2 18495.853} C_VEL
LIN {X 0,Y 423.567,Z 956.973,A -85,B 0,C 180,E1 18494.515,E2 18494.515} C_VEL
LIN {X 0,Y 419.977,Z 974.995,A -85,B 0,C 180,E1 18493.194,E2 18493.194} C_VEL
LIN {X 0,Y 415.535,Z 995.32,A -85,B 0,C 180,E1 18491.431,E2 18491.431} C_VEL
LIN {X 0,Y 411.247,Z 1013.364,A -85,B 0,C 180,E1 18489.569,E2 18489.569} C_VEL
LIN {X 0,Y 406.628,Z 1031.93,A -85,B 0,C 180,E1 18487.31,E2 18487.31} C_VEL
LIN {X 0,Y 404.234,Z 1041.241,A -85,B 0,C 180,E1 18486.031,E2 18486.031} C_VEL
LIN {X 0,Y 401.978,Z 1046.748,A -85,B 0,C 180,E1 18485.306,E2 18485.306} C_VEL
LIN {X 0,Y 393.233,Z 1060.555,A -85,B 0,C 180,E1 18483.605,E2 18483.605} C_VEL
LIN {X 0,Y 391.049,Z 1065.409,A -85,B 0,C 180,E1 18482.799,E2 18482.799} C_VEL
LIN {X 0,Y 387.166,Z 1079.881,A -85,B 0,C 180,E1 18479.896,E2 18479.896} C_VEL
LIN {X 0,Y 384.073,Z 1091.799,A -85,B 0,C 180,E1 18477.085,E2 18477.085} C_VEL
LIN {X 0,Y 381.139,Z 1104.106,A -85,B 0,C 180,E1 18473.664,E2 18473.664} C_VEL
LIN {X 0,Y 379.154,Z 1113.551,A -85,B 0,C 180,E1 18470.533,E2 18470.533} C_VEL
LIN {X 0,Y 377.644,Z 1122.076,A -85,B 0,C 180,E1 18467.091,E2 18467.091} C_VEL
LIN {X 0,Y 376.723,Z 1128.839,A -85,B 0,C 180,E1 18463.736,E2 18463.736} C_VEL
LIN {X 0,Y 376.205,Z 1133.925,A -85,B 0,C 180,E1 18460.413,E2 18460.413} C_VEL
LIN {X 0,Y 375.999,Z 1137.269,A -85,B 0,C 180,E1 18457.487,E2 18457.487} C_VEL
LIN {X 0,Y 375.933,Z 1139.849,A -85,B 0,C 180,E1 18453.966,E2 18453.966} C_VEL
LIN {X 0,Y 375.915,Z 1140.764,A -85,B 0,C 180,E1 18451.067,E2 18451.067} C_VEL
LIN {X 0,Y 375.926,Z 1140.625,A -85,B 0,C 180,E1 18447.866,E2 18447.866} C_VEL
LIN {X 0,Y 375.946,Z 1138.971,A -85,B 0,C 180,E1 18444.506,E2 18444.506} C_VEL
LIN {X 0,Y 376.073,Z 1136.277,A -85,B 0,C 180,E1 18441.438,E2 18441.438} C_VEL
LIN {X 0,Y 376.431,Z 1131.506,A -85,B 0,C 180,E1 18437.814,E2 18437.814} C_VEL
LIN {X 0,Y 377.089,Z 1125.905,A -85,B 0,C 180,E1 18434.624,E2 18434.624} C_VEL
LIN {X 0,Y 378.319,Z 1118.059,A -85,B 0,C 180,E1 18431.113,E2 18431.113} C_VEL
LIN {X 0,Y 380.081,Z 1109.089,A -85,B 0,C 180,E1 18427.818,E2 18427.818} C_VEL
LIN {X 0,Y 382.441,Z 1098.493,A -85,B 0,C 180,E1 18424.611,E2 18424.611} C_VEL
LIN {X 0,Y 385.468,Z 1086.437,A -85,B 0,C 180,E1 18421.493,E2 18421.493} C_VEL
LIN {X 0,Y 389.017,Z 1072.874,A -85,B 0,C 180,E1 18418.55,E2 18418.55} C_VEL
LIN {X 0,Y 393.329,Z 1057.176,A -85,B 0,C 180,E1 18415.644,E2 18415.644} C_VEL
LIN {X 0,Y 397.513,Z 1041.887,A -85,B 0,C 180,E1 18413.228,E2 18413.228} C_VEL
LIN {X 0,Y 402.254,Z 1024.218,A -85,B 0,C 180,E1 18410.85,E2 18410.85} C_VEL
LIN {X 0,Y 406.687,Z 1007.098,A -85,B 0,C 180,E1 18408.878,E2 18408.878} C_VEL
LIN {X 0,Y 411.296,Z 987.809,A -85,B 0,C 180,E1 18407,E2 18407} C_VEL
LIN {X 0,Y 415.663,Z 968.171,A -85,B 0,C 180,E1 18405.381,E2 18405.381} C_VEL
LIN {X 0,Y 419.659,Z 947.552,A -85,B 0,C 180,E1 18403.984,E2 18403.984} C_VEL
LIN {X 0,Y 423.36,Z 926.036,A -85,B 0,C 180,E1 18402.785,E2 18402.785} C_VEL
LIN {X 0,Y 426.316,Z 904.691,A -85,B 0,C 180,E1 18401.852,E2 18401.852} C_VEL
LIN {X 0,Y 428.887,Z 881.45,A -85,B 0,C 180,E1 18401.075,E2 18401.075} C_VEL
LIN {X 0,Y 430.484,Z 859.758,A -85,B 0,C 180,E1 18400.56,E2 18400.56} C_VEL
LIN {X 0,Y 439.373,Z 659.319,A -85,B 0,C 180,E1 18396.795,E2 18396.795} C_VEL
LIN {X 0,Y 441.267,Z 616.708,A -85,B 0,C 180,E1 18395.979,E2 18395.979} C_VEL
LIN {X 0,Y 431.593,Z 602.636,A -85,B 0,C 180,E1 18393.74,E2 18393.74} C_VEL
LIN {X 0,Y 421.67,Z 589.001,A -85,B 0,C 180,E1 18391.205,E2 18391.205} C_VEL
LIN {X 0,Y 412.833,Z 577.72,A -85,B 0,C 180,E1 18388.695,E2 18388.695} C_VEL
LIN {X 0,Y 408.827,Z 572.686,A -85,B 0,C 180,E1 18387.453,E2 18387.453} C_VEL
LIN {X 0,Y 404.501,Z 567.381,A -85,B 0,C 180,E1 18386.024,E2 18386.024} C_VEL
LIN {X 0,Y 400.927,Z 563.2,A -85,B 0,C 180,E1 18384.77,E2 18384.77} C_VEL
LIN {X 0,Y 399.67,Z 561.556,A -85,B 0,C 180,E1 18384.301,E2 18384.301} C_VEL
LIN {X 0,Y 396.209,Z 557.897,A -85,B 0,C 180,E1 18382.987,E2 18382.987} C_VEL
LIN {X 0,Y 394.663,Z 555.554,A -85,B 0,C 180,E1 18382.335,E2 18382.335} C_VEL
LIN {X 0,Y 391.264,Z 552.586,A -85,B 0,C 180,E1 18380.924,E2 18380.924} C_VEL
LIN {X 0,Y 389.308,Z 549.321,A -85,B 0,C 180,E1 18379.974,E2 18379.974} C_VEL
LIN {X 0,Y 386.008,Z 546.964,A -85,B 0,C 180,E1 18378.422,E2 18378.422} C_VEL
LIN {X 0,Y 383.994,Z 543.499,A -85,B 0,C 180,E1 18377.268,E2 18377.268} C_VEL
LIN {X 0,Y 383.51,Z 542.675,A -85,B 0,C 180,E1 18376.978,E2 18376.978} C_VEL
LIN {X 0,Y 379.955,Z 540.66,A -85,B 0,C 180,E1 18374.945,E2 18374.945} C_VEL
LIN {X 0,Y 378.068,Z 537.682,A -85,B 0,C 180,E1 18373.575,E2 18373.575} C_VEL
LIN {X 0,Y 377.657,Z 536,A -85,B 0,C 180,E1 18373.161,E2 18373.161} C_VEL
LIN {X 0,Y 377.661,Z 535.992,A -85,B 0,C 180,E1 18369.062,E2 18369.062} C_VEL
LIN {X 0,Y 377.67,Z 535.987,A -85,B 0,C 180,E1 18365.012,E2 18365.012} C_VEL
LIN {X 0,Y 377.678,Z 535.985,A -85,B 0,C 180,E1 18360.91,E2 18360.91} C_VEL
LIN {X 0,Y 377.679,Z 535.988,A -85,B 0,C 180,E1 18356.813,E2 18356.813} C_VEL
LIN {X 0,Y 377.688,Z 535.994,A -85,B 0,C 180,E1 18352.7,E2 18352.7} C_VEL
LIN {X 0,Y 377.672,Z 535.934,A -85,B 0,C 180,E1 18348.548,E2 18348.548} C_VEL
LIN {X 0,Y 377.703,Z 536.162,A -85,B 0,C 180,E1 18347.269,E2 18347.269} C_VEL
LIN {X 0,Y 378.598,Z 538.827,A -85,B 0,C 180,E1 18346.484,E2 18346.484} C_VEL
LIN {X 0,Y 380.916,Z 541.483,A -85,B 0,C 180,E1 18344.938,E2 18344.938} C_VEL
LIN {X 0,Y 383.798,Z 542.904,A -85,B 0,C 180,E1 18343.348,E2 18343.348} C_VEL
LIN {X 0,Y 385.36,Z 546.127,A -85,B 0,C 180,E1 18342.406,E2 18342.406} C_VEL
LIN {X 0,Y 388.388,Z 548.847,A -85,B 0,C 180,E1 18340.917,E2 18340.917} C_VEL
LIN {X 0,Y 389.638,Z 549.65,A -85,B 0,C 180,E1 18340.357,E2 18340.357} C_VEL
LIN {X 0,Y 391.834,Z 553.287,A -85,B 0,C 180,E1 18339.304,E2 18339.304} C_VEL
LIN {X 0,Y 395.19,Z 556.158,A -85,B 0,C 180,E1 18337.932,E2 18337.932} C_VEL
LIN {X 0,Y 398.043,Z 560.155,A -85,B 0,C 180,E1 18336.774,E2 18336.774} C_VEL
LIN {X 0,Y 400.513,Z 562.532,A -85,B 0,C 180,E1 18335.871,E2 18335.871} C_VEL
LIN {X 0,Y 403.935,Z 566.873,A -85,B 0,C 180,E1 18334.645,E2 18334.645} C_VEL
LIN {X 0,Y 408.686,Z 573.179,A -85,B 0,C 180,E1 18333.05,E2 18333.05} C_VEL
LIN {X 0,Y 413.902,Z 580.264,A -85,B 0,C 180,E1 18331.426,E2 18331.426} C_VEL
LIN {X 0,Y 422.175,Z 591.768,A -85,B 0,C 180,E1 18329.074,E2 18329.074} C_VEL
LIN {X 0,Y 431.665,Z 606.127,A -85,B 0,C 180,E1 18326.625,E2 18326.625} C_VEL
LIN {X 0,Y 440.845,Z 620.875,A -85,B 0,C 180,E1 18324.466,E2 18324.466} C_VEL
LIN {X 0,Y 441.435,Z 622.341,A -85,B 0,C 180,E1 18324.321,E2 18324.321} C_VEL
LIN {X 0,Y 431.856,Z 839.095,A -85,B 0,C 180,E1 18320.252,E2 18320.252} C_VEL
LIN {X 0,Y 429.431,Z 890.758,A -85,B 0,C 180,E1 18319.258,E2 18319.258} C_VEL
LIN {X 0,Y 427.124,Z 913.884,A -85,B 0,C 180,E1 18318.626,E2 18318.626} C_VEL
LIN {X 0,Y 424.271,Z 936.105,A -85,B 0,C 180,E1 18317.806,E2 18317.806} C_VEL
LIN {X 0,Y 420.978,Z 956.797,A -85,B 0,C 180,E1 18316.815,E2 18316.815} C_VEL
LIN {X 0,Y 416.96,Z 978.78,A -85,B 0,C 180,E1 18315.512,E2 18315.512} C_VEL
LIN {X 0,Y 412.957,Z 998.073,A -85,B 0,C 180,E1 18314.115,E2 18314.115} C_VEL
LIN {X 0,Y 408.212,Z 1019.105,A -85,B 0,C 180,E1 18312.294,E2 18312.294} C_VEL
LIN {X 0,Y 403.824,Z 1037.138,A -85,B 0,C 180,E1 18310.444,E2 18310.444} C_VEL
LIN {X 0,Y 398.973,Z 1056.12,A -85,B 0,C 180,E1 18308.152,E2 18308.152} C_VEL
LIN {X 0,Y 394.578,Z 1073.189,A -85,B 0,C 180,E1 18305.738,E2 18305.738} C_VEL
LIN {X 0,Y 390.356,Z 1089.26,A -85,B 0,C 180,E1 18303.064,E2 18303.064} C_VEL
LIN {X 0,Y 386.736,Z 1103.778,A -85,B 0,C 180,E1 18300.275,E2 18300.275} C_VEL
LIN {X 0,Y 383.505,Z 1117.118,A -85,B 0,C 180,E1 18297.248,E2 18297.248} C_VEL
LIN {X 0,Y 380.733,Z 1129.874,A -85,B 0,C 180,E1 18293.855,E2 18293.855} C_VEL
LIN {X 0,Y 378.936,Z 1139.35,A -85,B 0,C 180,E1 18290.867,E2 18290.867} C_VEL
LIN {X 0,Y 377.442,Z 1148.877,A -85,B 0,C 180,E1 18287.259,E2 18287.259} C_VEL
LIN {X 0,Y 376.638,Z 1155.575,A -85,B 0,C 180,E1 18284.136,E2 18284.136} C_VEL
LIN {X 0,Y 376.146,Z 1161.52,A -85,B 0,C 180,E1 18280.568,E2 18280.568} C_VEL
LIN {X 0,Y 375.967,Z 1165.11,A -85,B 0,C 180,E1 18277.641,E2 18277.641} C_VEL
LIN {X 0,Y 375.925,Z 1167.855,A -85,B 0,C 180,E1 18274.271,E2 18274.271} C_VEL
LIN {X 0,Y 375.917,Z 1168.936,A -85,B 0,C 180,E1 18271.219,E2 18271.219} C_VEL
LIN {X 0,Y 375.921,Z 1168.865,A -85,B 0,C 180,E1 18268.323,E2 18268.323} C_VEL
LIN {X 0,Y 375.927,Z 1167.237,A -85,B 0,C 180,E1 18264.811,E2 18264.811} C_VEL
LIN {X 0,Y 376.011,Z 1164.45,A -85,B 0,C 180,E1 18261.744,E2 18261.744} C_VEL
LIN {X 0,Y 376.28,Z 1159.672,A -85,B 0,C 180,E1 18258.193,E2 18258.193} C_VEL
LIN {X 0,Y 376.801,Z 1154.016,A -85,B 0,C 180,E1 18255.084,E2 18255.084} C_VEL
LIN {X 0,Y 377.835,Z 1146.226,A -85,B 0,C 180,E1 18251.644,E2 18251.644} C_VEL
LIN {X 0,Y 379.283,Z 1137.473,A -85,B 0,C 180,E1 18248.504,E2 18248.504} C_VEL
LIN {X 0,Y 381.557,Z 1125.993,A -85,B 0,C 180,E1 18245.045,E2 18245.045} C_VEL
LIN {X 0,Y 384.174,Z 1114.274,A -85,B 0,C 180,E1 18242.064,E2 18242.064} C_VEL
LIN {X 0,Y 387.654,Z 1099.88,A -85,B 0,C 180,E1 18238.945,E2 18238.945} C_VEL
LIN {X 0,Y 391.68,Z 1084.336,A -85,B 0,C 180,E1 18236.061,E2 18236.061} C_VEL
LIN {X 0,Y 395.872,Z 1068.03,A -85,B 0,C 180,E1 18233.501,E2 18233.501} C_VEL
LIN {X 0,Y 400.495,Z 1050.325,A -85,B 0,C 180,E1 18231.105,E2 18231.105} C_VEL
LIN {X 0,Y 404.896,Z 1032.726,A -85,B 0,C 180,E1 18229.081,E2 18229.081} C_VEL
LIN {X 0,Y 409.859,Z 1011.859,A -85,B 0,C 180,E1 18227.041,E2 18227.041} C_VEL
LIN {X 0,Y 414.132,Z 992.569,A -85,B 0,C 180,E1 18225.462,E2 18225.462} C_VEL
LIN {X 0,Y 418.422,Z 971.055,A -85,B 0,C 180,E1 18224.005,E2 18224.005} C_VEL
LIN {X 0,Y 421.998,Z 950.822,A -85,B 0,C 180,E1 18222.879,E2 18222.879} C_VEL
LIN {X 0,Y 425.321,Z 928.295,A -85,B 0,C 180,E1 18221.888,E2 18221.888} C_VEL
LIN {X 0,Y 427.759,Z 908.234,A -85,B 0,C 180,E1 18221.204,E2 18221.204} C_VEL
LIN {X 0,Y 429.792,Z 884.219,A -85,B 0,C 180,E1 18220.609,E2 18220.609} C_VEL
LIN {X 0,Y 438.146,Z 693.417,A -85,B 0,C 180,E1 18217.02,E2 18217.02} C_VEL
LIN {X 0,Y 441.302,Z 621.726,A -85,B 0,C 180,E1 18215.651,E2 18215.651} C_VEL
LIN {X 0,Y 432.329,Z 607.227,A -85,B 0,C 180,E1 18213.555,E2 18213.555} C_VEL
LIN {X 0,Y 423.909,Z 594.456,A -85,B 0,C 180,E1 18211.417,E2 18211.417} C_VEL
LIN {X 0,Y 415.107,Z 581.817,A -85,B 0,C 180,E1 18208.956,E2 18208.956} C_VEL
LIN {X 0,Y 406.925,Z 570.809,A -85,B 0,C 180,E1 18206.406,E2 18206.406} C_VEL
LIN {X 0,Y 402.874,Z 565.811,A -85,B 0,C 180,E1 18205.033,E2 18205.033} C_VEL
LIN {X 0,Y 399.595,Z 561.478,A -85,B 0,C 180,E1 18203.834,E2 18203.834} C_VEL
LIN {X 0,Y 396.212,Z 557.925,A -85,B 0,C 180,E1 18202.555,E2 18202.555} C_VEL
LIN {X 0,Y 394.93,Z 555.699,A -85,B 0,C 180,E1 18202.005,E2 18202.005} C_VEL
LIN {X 0,Y 391.561,Z 552.966,A -85,B 0,C 180,E1 18200.633,E2 18200.633} C_VEL
LIN {X 0,Y 389.528,Z 549.41,A -85,B 0,C 180,E1 18199.649,E2 18199.649} C_VEL
LIN {X 0,Y 386.044,Z 546.973,A -85,B 0,C 180,E1 18198.029,E2 18198.029} C_VEL
LIN {X 0,Y 384.063,Z 543.706,A -85,B 0,C 180,E1 18196.913,E2 18196.913} C_VEL
LIN {X 0,Y 383.666,Z 542.711,A -85,B 0,C 180,E1 18196.658,E2 18196.658} C_VEL
LIN {X 0,Y 380.172,Z 540.86,A -85,B 0,C 180,E1 18194.702,E2 18194.702} C_VEL
LIN {X 0,Y 378.175,Z 537.946,A -85,B 0,C 180,E1 18193.298,E2 18193.298} C_VEL
LIN {X 0,Y 377.673,Z 535.959,A -85,B 0,C 180,E1 18192.771,E2 18192.771} C_VEL
LIN {X 0,Y 377.674,Z 535.964,A -85,B 0,C 180,E1 18188.679,E2 18188.679} C_VEL
LIN {X 0,Y 377.677,Z 535.993,A -85,B 0,C 180,E1 18184.555,E2 18184.555} C_VEL
LIN {X 0,Y 377.684,Z 536.001,A -85,B 0,C 180,E1 18180.455,E2 18180.455} C_VEL
LIN {X 0,Y 377.682,Z 536.003,A -85,B 0,C 180,E1 18176.357,E2 18176.357} C_VEL
LIN {X 0,Y 377.685,Z 535.988,A -85,B 0,C 180,E1 18172.24,E2 18172.24} C_VEL
LIN {X 0,Y 377.679,Z 535.941,A -85,B 0,C 180,E1 18168.083,E2 18168.083} C_VEL
LIN {X 0,Y 377.687,Z 536.146,A -85,B 0,C 180,E1 18166.587,E2 18166.587} C_VEL
LIN {X 0,Y 378.62,Z 538.866,A -85,B 0,C 180,E1 18165.783,E2 18165.783} C_VEL
LIN {X 0,Y 380.85,Z 541.404,A -85,B 0,C 180,E1 18164.311,E2 18164.311} C_VEL
LIN {X 0,Y 383.81,Z 542.946,A -85,B 0,C 180,E1 18162.684,E2 18162.684} C_VEL
LIN {X 0,Y 385.569,Z 546.425,A -85,B 0,C 180,E1 18161.645,E2 18161.645} C_VEL
LIN {X 0,Y 388.362,Z 548.855,A -85,B 0,C 180,E1 18160.289,E2 18160.289} C_VEL
LIN {X 0,Y 389.613,Z 549.698,A -85,B 0,C 180,E1 18159.729,E2 18159.729} C_VEL
LIN {X 0,Y 391.829,Z 553.276,A -85,B 0,C 180,E1 18158.677,E2 18158.677} C_VEL
LIN {X 0,Y 395.199,Z 556.189,A -85,B 0,C 180,E1 18157.305,E2 18157.305} C_VEL
LIN {X 0,Y 398.068,Z 560.176,A -85,B 0,C 180,E1 18156.146,E2 18156.146} C_VEL
LIN {X 0,Y 400.458,Z 562.439,A -85,B 0,C 180,E1 18155.278,E2 18155.278} C_VEL
LIN {X 0,Y 403.787,Z 566.756,A -85,B 0,C 180,E1 18154.084,E2 18154.084} C_VEL
LIN {X 0,Y 405.646,Z 568.739,A -85,B 0,C 180,E1 18153.464,E2 18153.464} C_VEL
LIN {X 0,Y 409.547,Z 573.372,A -85,B 0,C 180,E1 18152.205,E2 18152.205} C_VEL
LIN {X 0,Y 418.991,Z 585.614,A -85,B 0,C 180,E1 18149.41,E2 18149.41} C_VEL
LIN {X 0,Y 426.517,Z 595.624,A -85,B 0,C 180,E1 18147.412,E2 18147.412} C_VEL
LIN {X 0,Y 435.913,Z 608.84,A -85,B 0,C 180,E1 18145.13,E2 18145.13} C_VEL
LIN {X 0,Y 441.311,Z 616.963,A -85,B 0,C 180,E1 18143.905,E2 18143.905} C_VEL
LIN {X 0,Y 431.983,Z 825.738,A -85,B 0,C 180,E1 18139.99,E2 18139.99} C_VEL
LIN {X 0,Y 429.817,Z 870.154,A -85,B 0,C 180,E1 18139.128,E2 18139.128} C_VEL
LIN {X 0,Y 427.69,Z 892.622,A -85,B 0,C 180,E1 18138.49,E2 18138.49} C_VEL
LIN {X 0,Y 424.839,Z 915.765,A -85,B 0,C 180,E1 18137.597,E2 18137.597} C_VEL
LIN {X 0,Y 421.829,Z 935.167,A -85,B 0,C 180,E1 18136.639,E2 18136.639} C_VEL
LIN {X 0,Y 417.816,Z 957.38,A -85,B 0,C 180,E1 18135.286,E2 18135.286} C_VEL
LIN {X 0,Y 414.095,Z 975.306,A -85,B 0,C 180,E1 18133.963,E2 18133.963} C_VEL
LIN {X 0,Y 409.459,Z 995.631,A -85,B 0,C 180,E1 18132.185,E2 18132.185} C_VEL
LIN {X 0,Y 404.966,Z 1013.676,A -85,B 0,C 180,E1 18130.307,E2 18130.307} C_VEL
LIN {X 0,Y 400.115,Z 1032.242,A -85,B 0,C 180,E1 18128.024,E2 18128.024} C_VEL
LIN {X 0,Y 395.759,Z 1048.355,A -85,B 0,C 180,E1 18125.705,E2 18125.705} C_VEL
LIN {X 0,Y 391.49,Z 1063.773,A -85,B 0,C 180,E1 18123.101,E2 18123.101} C_VEL
LIN {X 0,Y 391.049,Z 1065.409,A -85,B 0,C 180,E1 18122.799,E2 18122.799} C_VEL
LIN {X 0,Y 388.888,Z 1070.315,A -85,B 0,C 180,E1 18121.964,E2 18121.964} C_VEL
LIN {X 0,Y 380.274,Z 1082.364,A -85,B 0,C 180,E1 18119.936,E2 18119.936} C_VEL
LIN {X 0,Y 378.216,Z 1086.719,A -85,B 0,C 180,E1 18119.02,E2 18119.02} C_VEL
LIN {X 0,Y 374.913,Z 1099.062,A -85,B 0,C 180,E1 18115.767,E2 18115.767} C_VEL
LIN {X 0,Y 372.344,Z 1109.834,A -85,B 0,C 180,E1 18112.416,E2 18112.416} C_VEL
LIN {X 0,Y 370.485,Z 1118.728,A -85,B 0,C 180,E1 18109.06,E2 18109.06} C_VEL
LIN {X 0,Y 369.142,Z 1126.685,A -85,B 0,C 180,E1 18105.363,E2 18105.363} C_VEL
LIN {X 0,Y 368.452,Z 1132.278,A -85,B 0,C 180,E1 18102.061,E2 18102.061} C_VEL
LIN {X 0,Y 368.081,Z 1136.798,A -85,B 0,C 180,E1 18098.435,E2 18098.435} C_VEL
LIN {X 0,Y 367.954,Z 1139.427,A -85,B 0,C 180,E1 18095.301,E2 18095.301} C_VEL
LIN {X 0,Y 367.926,Z 1140.977,A -85,B 0,C 180,E1 18091.713,E2 18091.713} C_VEL
LIN {X 0,Y 367.921,Z 1141.055,A -85,B 0,C 180,E1 18088.755,E2 18088.755} C_VEL
LIN {X 0,Y 367.943,Z 1139.993,A -85,B 0,C 180,E1 18085.48,E2 18085.48} C_VEL
LIN {X 0,Y 368.044,Z 1137.352,A -85,B 0,C 180,E1 18082.036,E2 18082.036} C_VEL
LIN {X 0,Y 368.315,Z 1133.744,A -85,B 0,C 180,E1 18078.887,E2 18078.887} C_VEL
LIN {X 0,Y 368.952,Z 1127.976,A -85,B 0,C 180,E1 18075.242,E2 18075.242} C_VEL
